Yaskawa INFORM job: tourneTRJ2.JBI

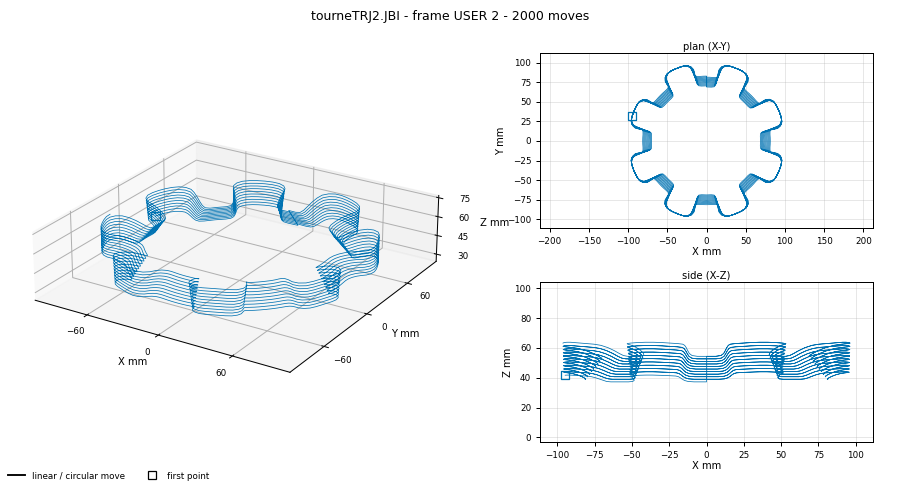
[picture p0: tool path of tourneTRJ2.JBI in frame USER 2, 2000 of 2000 moves have a stored position in this frame; points joined in program order, loops and branches not executed]
/JOB
//NAME tourneTRJ2
///FOLDERNAME DEMO
//POS
///NPOS 2000,0,2000,0,0,0
///USER 2
///TOOL 7
///POSTYPE USER
///RECTAN
///RCONF 1,0,0,0,0,0,0,0,0,0,0,0,0,0,0,0,0,0,0,0,0,0,0,0
C00000=-94.679,31.992,41.678,179.9348,0.0039,-7128.6701
C00001=-93.214,36.189,41.785,179.9926,-0.0033,-7131.2180
C00002=-91.502,40.323,41.785,179.9924,-0.0029,-7133.7821
C00003=-89.570,44.326,41.678,179.9359,-0.0003,-7136.3297
C00004=-87.153,47.905,41.515,178.5880,-0.3682,-7138.7961
C00005=-83.964,50.341,41.355,178.0736,-1.1845,-7140.9450
C00006=-80.606,51.270,41.159,177.8332,-3.2869,-7142.4587
C00007=-77.545,50.645,40.789,178.9173,-3.7322,-7143.1487
C00008=-74.511,49.565,40.048,179.7943,-0.8472,-7143.6320
C00009=-71.724,48.673,39.090,-178.2386,5.1754,-7144.1614
C00010=-69.261,48.447,38.165,-169.6493,15.1644,-7144.9722
C00011=-66.868,49.465,37.495,-147.2874,13.5004,-7146.4919
C00012=-64.059,52.288,37.229,-142.4203,2.3568,-7149.2230
C00013=-61.349,55.398,37.217,-142.1949,-0.1576,-7152.0820
C00014=-58.451,58.451,37.225,-142.2074,0.0000,-7155.0000
C00015=-55.398,61.349,37.217,-142.1949,0.1576,-7157.9180
C00016=-52.288,64.059,37.229,-142.4203,-2.3568,-7160.7770
C00017=-49.465,66.868,37.495,-147.2834,-13.4965,-7163.5081
C00018=-48.447,69.261,38.165,-169.6493,-15.1644,-7165.0278
C00019=-48.673,71.724,39.090,-178.2386,-5.1754,-7165.8386
C00020=-49.565,74.511,40.048,179.7943,0.8472,-7166.3680
C00021=-50.645,77.545,40.789,178.9173,3.7322,-7166.8513
C00022=-51.270,80.606,41.159,177.8332,3.2869,-7167.5413
C00023=-50.341,83.964,41.355,178.0736,1.1845,-7169.0550
C00024=-47.905,87.153,41.515,178.5880,0.3682,-7171.2039
C00025=-44.326,89.570,41.678,179.9359,0.0003,-7173.6703
C00026=-40.323,91.502,41.785,179.9924,0.0029,-7176.2179
C00027=-36.189,93.214,41.785,179.9926,0.0033,-7178.7820
C00028=-31.992,94.679,41.678,179.9348,-0.0039,-7181.3299
C00029=-27.752,95.500,41.515,178.5912,-0.3677,-7183.7963
C00030=-23.775,94.968,41.355,178.0749,-1.1854,-7185.9450
C00031=-20.743,93.250,41.159,177.8320,-3.2854,-7187.4590
C00032=-19.021,90.644,40.789,178.9181,-3.7308,-7188.1488
C00033=-17.640,87.735,40.048,179.7952,-0.8419,-7188.6317
C00034=-16.299,85.134,39.090,-178.2398,5.1751,-7189.1618
C00035=-14.718,83.232,38.165,-169.6494,15.1618,-7189.9720
C00036=-12.305,82.260,37.495,-147.2854,13.4971,-7191.4924
C00037=-8.324,82.270,37.229,-142.4221,2.3584,-7194.2225
C00038=-4.208,82.553,37.217,-142.1936,-0.1593,-7197.0820
C00039=0.000,82.662,37.225,-142.2064,0.0000,-7200.0000
C00040=0.000,81.307,38.958,-141.7572,0.0000,-7200.0000
C00041=4.084,81.202,38.949,-141.7490,0.1755,-7202.8792
C00042=8.115,80.931,38.962,-141.9996,-2.6222,-7205.7259
C00043=12.050,80.963,39.253,-147.5601,-14.5903,-7208.4654
C00044=14.402,82.041,39.987,-171.3983,-14.2979,-7209.9566
C00045=15.932,84.113,41.004,-178.8180,-4.0002,-7210.7254
C00046=17.234,86.943,42.060,179.6316,1.7672,-7211.2119
C00047=18.580,90.119,42.880,178.8638,4.5859,-7211.6495
C00048=20.259,92.987,43.289,177.5830,4.0974,-7212.2909
C00049=23.317,94.913,43.506,177.7331,1.4901,-7213.8024
C00050=27.389,95.566,43.684,178.4237,0.4280,-7215.9922
C00051=31.762,94.755,43.864,179.9221,0.0019,-7218.5312
C00052=36.110,93.244,43.984,179.9872,-0.0012,-7221.1696
C00053=40.400,91.468,43.984,179.9872,-0.0006,-7223.8303
C00054=44.543,89.461,43.864,179.9231,-0.0001,-7226.4689
C00055=48.209,86.942,43.684,178.4246,-0.4305,-7229.0082
C00056=50.626,83.601,43.506,177.7365,-1.4915,-7231.1977
C00057=51.426,80.077,43.289,177.5870,-4.0930,-7232.7089
C00058=50.586,76.861,42.880,178.8633,-4.5829,-7233.3509
C00059=49.291,73.664,42.060,179.6313,-1.7668,-7233.7878
C00060=48.211,70.742,41.004,-178.8201,3.9998,-7234.2746
C00061=47.828,68.195,39.987,-171.4011,14.2972,-7235.0436
C00062=48.729,65.770,39.253,-147.5575,14.5879,-7236.5348
C00063=51.488,62.965,38.962,-141.9986,2.6207,-7239.2737
C00064=54.531,60.307,38.949,-141.7481,-0.1713,-7242.1206
C00065=57.493,57.493,38.958,-141.7571,0.0000,-7245.0000
C00066=60.306,54.531,38.949,-141.7481,0.1717,-7247.8789
C00067=62.965,51.488,38.962,-141.9986,-2.6207,-7250.7263
C00068=65.770,48.729,39.253,-147.5575,-14.5879,-7253.4652
C00069=68.195,47.828,39.987,-171.4011,-14.2972,-7254.9564
C00070=70.742,48.211,41.004,-178.8201,-3.9998,-7255.7254
C00071=73.664,49.291,42.060,179.6313,1.7668,-7256.2122
C00072=76.861,50.586,42.880,178.8633,4.5829,-7256.6491
C00073=80.077,51.426,43.289,177.5870,4.0930,-7257.2911
C00074=83.601,50.626,43.506,177.7365,1.4915,-7258.8023
C00075=86.942,48.209,43.684,178.4246,0.4305,-7260.9918
C00076=89.461,44.543,43.864,179.9231,0.0001,-7263.5311
C00077=91.468,40.400,43.984,179.9872,0.0006,-7266.1697
C00078=93.244,36.110,43.984,179.9872,0.0012,-7268.8304
C00079=94.755,31.762,43.864,179.9221,-0.0019,-7271.4688
C00080=95.566,27.389,43.684,178.4237,-0.4280,-7274.0078
C00081=94.913,23.317,43.506,177.7331,-1.4901,-7276.1976
C00082=92.987,20.259,43.289,177.5830,-4.0974,-7277.7091
C00083=90.119,18.580,42.880,178.8638,-4.5859,-7278.3505
C00084=86.943,17.234,42.060,179.6316,-1.7672,-7278.7881
C00085=84.113,15.932,41.004,-178.8180,4.0002,-7279.2746
C00086=82.041,14.402,39.987,-171.3983,14.2979,-7280.0434
C00087=80.963,12.050,39.253,-147.5601,14.5903,-7281.5346
C00088=80.931,8.115,38.962,-141.9996,2.6222,-7284.2741
C00089=81.202,4.084,38.949,-141.7490,-0.1755,-7287.1208
C00090=81.307,0.000,38.958,-141.7572,-0.0000,-7290.0000
C00091=81.202,-4.084,38.949,-141.7490,0.1755,-7292.8792
C00092=80.931,-8.116,38.962,-141.9996,-2.6227,-7295.7266
C00093=80.963,-12.050,39.253,-147.5601,-14.5903,-7298.4654
C00094=82.041,-14.402,39.987,-171.3983,-14.2979,-7299.9566
C00095=84.113,-15.932,41.004,-178.8180,-4.0002,-7300.7254
C00096=86.943,-17.234,42.060,179.6316,1.7672,-7301.2119
C00097=90.119,-18.580,42.880,178.8638,4.5859,-7301.6495
C00098=92.987,-20.259,43.289,177.5830,4.0974,-7302.2909
C00099=94.913,-23.317,43.506,177.7331,1.4901,-7303.8024
C00100=95.566,-27.389,43.684,178.4237,0.4280,-7305.9922
C00101=94.755,-31.762,43.864,179.9221,0.0019,-7308.5312
C00102=93.244,-36.110,43.984,179.9872,-0.0012,-7311.1696
C00103=91.468,-40.400,43.984,179.9872,-0.0006,-7313.8303
C00104=89.461,-44.543,43.864,179.9231,-0.0001,-7316.4689
C00105=86.942,-48.209,43.684,178.4246,-0.4305,-7319.0082
C00106=83.601,-50.626,43.506,177.7365,-1.4915,-7321.1977
C00107=80.077,-51.426,43.289,177.5870,-4.0930,-7322.7089
C00108=76.861,-50.586,42.880,178.8633,-4.5829,-7323.3509
C00109=73.664,-49.291,42.060,179.6313,-1.7668,-7323.7878
C00110=70.742,-48.211,41.004,-178.8201,3.9998,-7324.2746
C00111=68.195,-47.828,39.987,-171.4011,14.2972,-7325.0436
C00112=65.770,-48.729,39.253,-147.5575,14.5879,-7326.5348
C00113=62.965,-51.488,38.962,-141.9986,2.6207,-7329.2737
C00114=60.307,-54.531,38.949,-141.7481,-0.1713,-7332.1206
C00115=57.493,-57.493,38.958,-141.7571,0.0000,-7335.0000
C00116=54.531,-60.306,38.949,-141.7481,0.1717,-7337.8789
C00117=51.488,-62.965,38.962,-141.9986,-2.6207,-7340.7263
C00118=48.729,-65.770,39.253,-147.5575,-14.5879,-7343.4652
C00119=47.828,-68.195,39.987,-171.4011,-14.2972,-7344.9564
C00120=48.211,-70.742,41.004,-178.8201,-3.9998,-7345.7254
C00121=49.291,-73.664,42.060,179.6313,1.7668,-7346.2122
C00122=50.586,-76.861,42.880,178.8633,4.5829,-7346.6491
C00123=51.426,-80.077,43.289,177.5870,4.0930,-7347.2911
C00124=50.626,-83.601,43.506,177.7365,1.4915,-7348.8023
C00125=48.209,-86.942,43.684,178.4246,0.4305,-7350.9918
C00126=44.543,-89.461,43.864,179.9231,0.0001,-7353.5311
C00127=40.400,-91.468,43.984,179.9872,0.0006,-7356.1697
C00128=36.110,-93.244,43.984,179.9872,0.0012,-7358.8304
C00129=31.762,-94.755,43.864,179.9221,-0.0019,-7361.4688
C00130=27.389,-95.566,43.684,178.4237,-0.4280,-7364.0078
C00131=23.317,-94.913,43.506,177.7331,-1.4901,-7366.1976
C00132=20.259,-92.987,43.289,177.5830,-4.0974,-7367.7091
C00133=18.580,-90.119,42.880,178.8638,-4.5859,-7368.3505
C00134=17.234,-86.943,42.060,179.6316,-1.7672,-7368.7881
C00135=15.932,-84.113,41.004,-178.8180,4.0002,-7369.2746
C00136=14.402,-82.041,39.987,-171.3983,14.2979,-7370.0434
C00137=12.050,-80.963,39.253,-147.5601,14.5903,-7371.5346
C00138=8.115,-80.931,38.962,-141.9996,2.6222,-7374.2741
C00139=4.084,-81.202,38.949,-141.7490,-0.1755,-7377.1208
C00140=0.000,-81.307,38.958,-141.7572,0.0000,-7380.0000
C00141=0.000,-81.307,38.958,-141.7572,0.0000,-7380.0000
C00142=-4.084,-81.202,38.949,-141.7490,0.1755,-7382.8792
C00143=-8.116,-80.931,38.962,-141.9996,-2.6227,-7385.7266
C00144=-12.050,-80.963,39.253,-147.5601,-14.5903,-7388.4654
C00145=-14.402,-82.041,39.987,-171.3983,-14.2979,-7389.9566
C00146=-15.932,-84.113,41.004,-178.8180,-4.0002,-7390.7254
C00147=-17.234,-86.943,42.060,179.6316,1.7672,-7391.2119
C00148=-18.580,-90.119,42.880,178.8638,4.5859,-7391.6495
C00149=-20.259,-92.987,43.289,177.5830,4.0974,-7392.2909
C00150=-23.317,-94.913,43.506,177.7331,1.4901,-7393.8024
C00151=-27.389,-95.566,43.684,178.4237,0.4280,-7395.9922
C00152=-31.762,-94.755,43.864,179.9221,0.0019,-7398.5312
C00153=-36.110,-93.244,43.984,179.9872,-0.0012,-7401.1696
C00154=-40.400,-91.468,43.984,179.9872,-0.0006,-7403.8303
C00155=-44.543,-89.461,43.864,179.9231,-0.0001,-7406.4689
C00156=-48.209,-86.942,43.684,178.4246,-0.4305,-7409.0082
C00157=-50.626,-83.601,43.506,177.7365,-1.4915,-7411.1977
C00158=-51.426,-80.077,43.289,177.5870,-4.0930,-7412.7089
C00159=-50.586,-76.861,42.880,178.8633,-4.5829,-7413.3509
C00160=-49.291,-73.664,42.060,179.6313,-1.7668,-7413.7878
C00161=-48.211,-70.742,41.004,-178.8201,3.9998,-7414.2746
C00162=-47.828,-68.195,39.987,-171.4011,14.2972,-7415.0436
C00163=-48.729,-65.770,39.253,-147.5575,14.5879,-7416.5348
C00164=-51.488,-62.965,38.962,-141.9986,2.6207,-7419.2737
C00165=-54.531,-60.307,38.949,-141.7481,-0.1713,-7422.1206
C00166=-57.493,-57.493,38.958,-141.7571,-0.0000,-7425.0000
C00167=-60.306,-54.531,38.949,-141.7481,0.1717,-7427.8789
C00168=-62.965,-51.488,38.962,-141.9986,-2.6207,-7430.7263
C00169=-65.770,-48.729,39.253,-147.5575,-14.5879,-7433.4652
C00170=-68.195,-47.828,39.987,-171.4011,-14.2972,-7434.9564
C00171=-70.742,-48.211,41.004,-178.8201,-3.9998,-7435.7254
C00172=-73.664,-49.291,42.060,179.6313,1.7668,-7436.2122
C00173=-76.861,-50.586,42.880,178.8633,4.5829,-7436.6491
C00174=-80.077,-51.426,43.289,177.5870,4.0930,-7437.2911
C00175=-83.601,-50.626,43.506,177.7365,1.4915,-7438.8023
C00176=-86.942,-48.209,43.684,178.4246,0.4305,-7440.9918
C00177=-89.461,-44.543,43.864,179.9231,0.0001,-7443.5311
C00178=-91.468,-40.400,43.984,179.9872,0.0006,-7446.1697
C00179=-93.244,-36.110,43.984,179.9872,0.0012,-7448.8304
C00180=-94.755,-31.762,43.864,179.9221,-0.0019,-7451.4688
C00181=-95.566,-27.389,43.684,178.4237,-0.4280,-7454.0078
C00182=-94.913,-23.317,43.506,177.7331,-1.4901,-7456.1976
C00183=-92.987,-20.259,43.289,177.5830,-4.0974,-7457.7091
C00184=-90.119,-18.580,42.880,178.8638,-4.5859,-7458.3505
C00185=-86.943,-17.234,42.060,179.6316,-1.7672,-7458.7881
C00186=-84.113,-15.932,41.004,-178.8180,4.0002,-7459.2746
C00187=-82.041,-14.402,39.987,-171.3983,14.2979,-7460.0434
C00188=-80.963,-12.050,39.253,-147.5601,14.5903,-7461.5346
C00189=-80.931,-8.115,38.962,-141.9996,2.6222,-7464.2741
C00190=-81.202,-4.084,38.949,-141.7490,-0.1755,-7467.1208
C00191=-81.307,0.000,38.958,-141.7572,-0.0000,-7470.0000
C00192=-81.202,4.084,38.949,-141.7490,0.1755,-7472.8792
C00193=-80.931,8.116,38.962,-141.9996,-2.6227,-7475.7266
C00194=-80.963,12.050,39.253,-147.5601,-14.5903,-7478.4654
C00195=-82.041,14.402,39.987,-171.3983,-14.2979,-7479.9566
C00196=-84.113,15.932,41.004,-178.8180,-4.0002,-7480.7254
C00197=-86.943,17.234,42.060,179.6316,1.7672,-7481.2119
C00198=-90.119,18.580,42.880,178.8638,4.5859,-7481.6495
C00199=-92.987,20.259,43.289,177.5830,4.0974,-7482.2909
C00200=-94.913,23.317,43.506,177.7331,1.4901,-7483.8024
C00201=-95.566,27.389,43.684,178.4237,0.4280,-7485.9922
C00202=-94.755,31.762,43.864,179.9221,0.0019,-7488.5312
C00203=-93.244,36.110,43.984,179.9872,-0.0012,-7491.1696
C00204=-91.468,40.400,43.984,179.9872,-0.0006,-7493.8303
C00205=-89.461,44.543,43.864,179.9231,-0.0001,-7496.4689
C00206=-86.942,48.209,43.684,178.4246,-0.4305,-7499.0082
C00207=-83.601,50.626,43.506,177.7365,-1.4915,-7501.1977
C00208=-80.077,51.426,43.289,177.5870,-4.0930,-7502.7089
C00209=-76.861,50.586,42.880,178.8633,-4.5829,-7503.3509
C00210=-73.664,49.291,42.060,179.6313,-1.7668,-7503.7878
C00211=-70.742,48.211,41.004,-178.8201,3.9998,-7504.2746
C00212=-68.195,47.828,39.987,-171.4011,14.2972,-7505.0436
C00213=-65.770,48.729,39.253,-147.5575,14.5879,-7506.5348
C00214=-62.965,51.488,38.962,-141.9986,2.6207,-7509.2737
C00215=-60.307,54.531,38.949,-141.7481,-0.1713,-7512.1206
C00216=-57.493,57.493,38.958,-141.7571,-0.0000,-7515.0000
C00217=-54.531,60.306,38.949,-141.7481,0.1717,-7517.8789
C00218=-51.488,62.965,38.962,-141.9986,-2.6207,-7520.7263
C00219=-48.729,65.770,39.253,-147.5575,-14.5879,-7523.4652
C00220=-47.828,68.195,39.987,-171.4011,-14.2972,-7524.9564
C00221=-48.211,70.742,41.004,-178.8201,-3.9998,-7525.7254
C00222=-49.291,73.664,42.060,179.6313,1.7668,-7526.2122
C00223=-50.586,76.861,42.880,178.8633,4.5829,-7526.6491
C00224=-51.426,80.077,43.289,177.5870,4.0930,-7527.2911
C00225=-50.626,83.601,43.506,177.7365,1.4915,-7528.8023
C00226=-48.209,86.942,43.684,178.4246,0.4305,-7530.9918
C00227=-44.543,89.461,43.864,179.9231,0.0001,-7533.5311
C00228=-40.400,91.468,43.984,179.9872,0.0006,-7536.1697
C00229=-36.110,93.244,43.984,179.9872,0.0012,-7538.8304
C00230=-31.762,94.755,43.864,179.9221,-0.0019,-7541.4688
C00231=-27.389,95.566,43.684,178.4237,-0.4280,-7544.0078
C00232=-23.317,94.913,43.506,177.7331,-1.4901,-7546.1976
C00233=-20.259,92.987,43.289,177.5830,-4.0974,-7547.7091
C00234=-18.580,90.119,42.880,178.8638,-4.5859,-7548.3505
C00235=-17.234,86.943,42.060,179.6316,-1.7672,-7548.7881
C00236=-15.932,84.113,41.004,-178.8180,4.0002,-7549.2746
C00237=-14.402,82.041,39.987,-171.3983,14.2979,-7550.0434
C00238=-12.050,80.963,39.253,-147.5601,14.5903,-7551.5346
C00239=-8.116,80.931,38.962,-141.9996,2.6227,-7554.2734
C00240=-4.084,81.202,38.949,-141.7490,-0.1755,-7557.1208
C00241=0.000,81.307,38.958,-141.7572,-0.0000,-7560.0000
C00242=0.000,79.940,40.681,-141.3939,-0.0000,-7560.0000
C00243=3.959,79.840,40.672,-141.3825,0.1903,-7562.8388
C00244=7.905,79.580,40.686,-141.6632,-2.8895,-7565.6728
C00245=11.791,79.654,41.003,-147.9831,-15.6038,-7568.4202
C00246=14.083,80.839,41.802,-172.9728,-13.2411,-7569.8823
C00247=15.561,83.082,42.912,-179.2626,-2.8848,-7570.6084
C00248=16.825,86.143,44.068,179.5316,2.5969,-7571.0516
C00249=18.134,89.588,44.968,178.8691,5.3340,-7571.4429
C00250=19.771,92.721,45.418,177.4283,4.8395,-7572.0370
C00251=22.856,94.857,45.657,177.4311,1.7993,-7573.5473
C00252=27.022,95.633,45.852,178.2699,0.4949,-7575.7781
C00253=31.529,94.831,46.051,179.9040,0.0017,-7578.3907
C00254=36.031,93.275,46.182,179.9872,-0.0012,-7581.1209
C00255=40.478,91.433,46.182,179.9872,-0.0006,-7583.8793
C00256=44.762,89.350,46.051,179.9026,-0.0025,-7586.6097
C00257=48.515,86.730,45.852,178.2708,-0.4972,-7589.2218
C00258=50.913,83.236,45.657,177.4345,-1.7991,-7591.4529
C00259=51.583,79.544,45.418,177.4322,-4.8395,-7592.9628
C00260=50.526,76.172,44.968,178.8696,-5.3331,-7593.5569
C00261=49.015,72.810,44.068,179.5365,-2.5972,-7593.9481
C00262=47.744,69.752,42.912,-179.2614,2.8847,-7594.3909
C00263=47.203,67.120,41.802,-172.9761,13.2392,-7595.1173
C00264=47.986,64.662,41.003,-147.9821,15.6031,-7596.5793
C00265=50.682,61.862,40.686,-141.6667,2.8929,-7599.3269
C00266=53.655,59.255,40.672,-141.3805,-0.1909,-7602.1606
C00267=56.526,56.526,40.681,-141.3961,0.0000,-7605.0000
C00268=59.255,53.656,40.672,-141.3805,0.1913,-7607.8388
C00269=61.862,50.682,40.686,-141.6667,-2.8929,-7610.6731
C00270=64.662,47.986,41.003,-147.9821,-15.6031,-7613.4207
C00271=67.120,47.203,41.802,-172.9761,-13.2392,-7614.8827
C00272=69.752,47.744,42.912,-179.2614,-2.8847,-7615.6091
C00273=72.810,49.015,44.068,179.5365,2.5972,-7616.0519
C00274=76.172,50.526,44.968,178.8696,5.3331,-7616.4431
C00275=79.544,51.583,45.418,177.4322,4.8395,-7617.0372
C00276=83.236,50.913,45.657,177.4345,1.7991,-7618.5471
C00277=86.730,48.515,45.852,178.2708,0.4972,-7620.7782
C00278=89.350,44.762,46.051,179.9026,0.0025,-7623.3903
C00279=91.433,40.478,46.182,179.9872,0.0006,-7626.1207
C00280=93.275,36.031,46.182,179.9872,0.0012,-7628.8791
C00281=94.831,31.529,46.051,179.9040,-0.0017,-7631.6093
C00282=95.633,27.022,45.852,178.2699,-0.4949,-7634.2219
C00283=94.857,22.856,45.657,177.4311,-1.7993,-7636.4527
C00284=92.721,19.771,45.418,177.4283,-4.8395,-7637.9630
C00285=89.588,18.134,44.968,178.8691,-5.3340,-7638.5571
C00286=86.143,16.825,44.068,179.5316,-2.5969,-7638.9484
C00287=83.082,15.561,42.912,-179.2626,2.8848,-7639.3916
C00288=80.839,14.083,41.802,-172.9728,13.2411,-7640.1177
C00289=79.654,11.791,41.003,-147.9831,15.6038,-7641.5798
C00290=79.580,7.905,40.686,-141.6632,2.8895,-7644.3272
C00291=79.840,3.959,40.672,-141.3825,-0.1903,-7647.1612
C00292=79.940,0.000,40.681,-141.3939,0.0000,-7650.0000
C00293=79.840,-3.959,40.672,-141.3825,0.1903,-7652.8388
C00294=79.580,-7.905,40.686,-141.6677,-2.8888,-7655.6728
C00295=79.654,-11.792,41.003,-147.9832,-15.6042,-7658.4209
C00296=80.839,-14.083,41.802,-172.9728,-13.2411,-7659.8823
C00297=83.082,-15.561,42.912,-179.2626,-2.8848,-7660.6084
C00298=86.143,-16.825,44.068,179.5316,2.5969,-7661.0516
C00299=89.588,-18.134,44.968,178.8691,5.3340,-7661.4429
C00300=92.721,-19.771,45.418,177.4283,4.8395,-7662.0370
C00301=94.857,-22.856,45.657,177.4311,1.7993,-7663.5473
C00302=95.633,-27.022,45.852,178.2699,0.4949,-7665.7781
C00303=94.831,-31.529,46.051,179.9040,0.0017,-7668.3907
C00304=93.275,-36.031,46.182,179.9872,-0.0012,-7671.1209
C00305=91.433,-40.478,46.182,179.9872,-0.0006,-7673.8793
C00306=89.350,-44.762,46.051,179.9026,-0.0025,-7676.6097
C00307=86.730,-48.515,45.852,178.2708,-0.4972,-7679.2218
C00308=83.236,-50.913,45.657,177.4345,-1.7991,-7681.4529
C00309=79.544,-51.583,45.418,177.4322,-4.8395,-7682.9628
C00310=76.172,-50.526,44.968,178.8696,-5.3331,-7683.5569
C00311=72.810,-49.015,44.068,179.5365,-2.5972,-7683.9481
C00312=69.752,-47.744,42.912,-179.2614,2.8847,-7684.3909
C00313=67.120,-47.203,41.802,-172.9761,13.2392,-7685.1173
C00314=64.662,-47.986,41.003,-147.9821,15.6031,-7686.5793
C00315=61.862,-50.682,40.686,-141.6667,2.8929,-7689.3269
C00316=59.255,-53.655,40.672,-141.3805,-0.1909,-7692.1606
C00317=56.526,-56.526,40.681,-141.3961,0.0000,-7695.0000
C00318=53.656,-59.255,40.672,-141.3805,0.1913,-7697.8388
C00319=50.682,-61.862,40.686,-141.6667,-2.8929,-7700.6731
C00320=47.986,-64.662,41.003,-147.9821,-15.6031,-7703.4207
C00321=47.203,-67.120,41.802,-172.9761,-13.2392,-7704.8827
C00322=47.744,-69.752,42.912,-179.2614,-2.8847,-7705.6091
C00323=49.015,-72.810,44.068,179.5365,2.5972,-7706.0519
C00324=50.526,-76.172,44.968,178.8696,5.3331,-7706.4431
C00325=51.583,-79.544,45.418,177.4322,4.8395,-7707.0372
C00326=50.913,-83.236,45.657,177.4345,1.7991,-7708.5471
C00327=48.515,-86.730,45.852,178.2708,0.4972,-7710.7782
C00328=44.762,-89.350,46.051,179.9026,0.0025,-7713.3903
C00329=40.478,-91.433,46.182,179.9872,0.0006,-7716.1207
C00330=36.031,-93.275,46.182,179.9872,0.0012,-7718.8791
C00331=31.529,-94.831,46.051,179.9040,-0.0017,-7721.6093
C00332=27.022,-95.633,45.852,178.2699,-0.4949,-7724.2219
C00333=22.856,-94.857,45.657,177.4311,-1.7993,-7726.4527
C00334=19.771,-92.721,45.418,177.4283,-4.8395,-7727.9630
C00335=18.134,-89.588,44.968,178.8691,-5.3340,-7728.5571
C00336=16.825,-86.143,44.068,179.5316,-2.5969,-7728.9484
C00337=15.561,-83.082,42.912,-179.2626,2.8848,-7729.3916
C00338=14.083,-80.839,41.802,-172.9728,13.2411,-7730.1177
C00339=11.791,-79.654,41.003,-147.9831,15.6038,-7731.5798
C00340=7.905,-79.580,40.686,-141.6632,2.8895,-7734.3272
C00341=3.959,-79.840,40.672,-141.3825,-0.1903,-7737.1612
C00342=0.000,-79.940,40.681,-141.3939,0.0000,-7740.0000
C00343=0.000,-79.940,40.681,-141.3939,0.0000,-7740.0000
C00344=-3.959,-79.840,40.672,-141.3825,0.1903,-7742.8388
C00345=-7.905,-79.580,40.686,-141.6677,-2.8888,-7745.6728
C00346=-11.792,-79.654,41.003,-147.9832,-15.6042,-7748.4209
C00347=-14.083,-80.839,41.802,-172.9728,-13.2411,-7749.8823
C00348=-15.561,-83.082,42.912,-179.2626,-2.8848,-7750.6084
C00349=-16.825,-86.143,44.068,179.5316,2.5969,-7751.0516
C00350=-18.134,-89.588,44.968,178.8691,5.3340,-7751.4429
C00351=-19.771,-92.721,45.418,177.4283,4.8395,-7752.0370
C00352=-22.856,-94.857,45.657,177.4311,1.7993,-7753.5473
C00353=-27.022,-95.633,45.852,178.2699,0.4949,-7755.7781
C00354=-31.529,-94.831,46.051,179.9040,0.0017,-7758.3907
C00355=-36.031,-93.275,46.182,179.9872,-0.0012,-7761.1209
C00356=-40.478,-91.433,46.182,179.9872,-0.0006,-7763.8793
C00357=-44.762,-89.350,46.051,179.9026,-0.0025,-7766.6097
C00358=-48.515,-86.730,45.852,178.2708,-0.4972,-7769.2218
C00359=-50.913,-83.236,45.657,177.4345,-1.7991,-7771.4529
C00360=-51.583,-79.544,45.418,177.4322,-4.8395,-7772.9628
C00361=-50.526,-76.172,44.968,178.8696,-5.3331,-7773.5569
C00362=-49.015,-72.810,44.068,179.5365,-2.5972,-7773.9481
C00363=-47.744,-69.752,42.912,-179.2614,2.8847,-7774.3909
C00364=-47.203,-67.120,41.802,-172.9761,13.2392,-7775.1173
C00365=-47.986,-64.662,41.003,-147.9821,15.6031,-7776.5793
C00366=-50.682,-61.862,40.686,-141.6667,2.8929,-7779.3269
C00367=-53.655,-59.255,40.672,-141.3805,-0.1909,-7782.1606
C00368=-56.526,-56.526,40.681,-141.3961,0.0000,-7785.0000
C00369=-59.255,-53.656,40.672,-141.3805,0.1913,-7787.8388
C00370=-61.862,-50.682,40.686,-141.6667,-2.8929,-7790.6731
C00371=-64.662,-47.986,41.003,-147.9821,-15.6031,-7793.4207
C00372=-67.120,-47.203,41.802,-172.9761,-13.2392,-7794.8827
C00373=-69.752,-47.744,42.912,-179.2614,-2.8847,-7795.6091
C00374=-72.810,-49.015,44.068,179.5365,2.5972,-7796.0519
C00375=-76.172,-50.526,44.968,178.8696,5.3331,-7796.4431
C00376=-79.544,-51.583,45.418,177.4322,4.8395,-7797.0372
C00377=-83.236,-50.913,45.657,177.4345,1.7991,-7798.5471
C00378=-86.730,-48.515,45.852,178.2708,0.4972,-7800.7782
C00379=-89.350,-44.762,46.051,179.9026,0.0025,-7803.3903
C00380=-91.433,-40.478,46.182,179.9872,0.0006,-7806.1207
C00381=-93.275,-36.031,46.182,179.9872,0.0012,-7808.8791
C00382=-94.831,-31.529,46.051,179.9040,-0.0017,-7811.6093
C00383=-95.633,-27.022,45.852,178.2699,-0.4949,-7814.2219
C00384=-94.857,-22.856,45.657,177.4311,-1.7993,-7816.4527
C00385=-92.721,-19.771,45.418,177.4283,-4.8395,-7817.9630
C00386=-89.588,-18.134,44.968,178.8691,-5.3340,-7818.5571
C00387=-86.143,-16.825,44.068,179.5316,-2.5969,-7818.9484
C00388=-83.082,-15.561,42.912,-179.2626,2.8848,-7819.3916
C00389=-80.839,-14.083,41.802,-172.9728,13.2411,-7820.1177
C00390=-79.654,-11.791,41.003,-147.9831,15.6038,-7821.5798
C00391=-79.580,-7.905,40.686,-141.6632,2.8895,-7824.3272
C00392=-79.840,-3.959,40.672,-141.3825,-0.1903,-7827.1612
C00393=-79.940,0.000,40.681,-141.3939,0.0000,-7830.0000
C00394=-79.840,3.959,40.672,-141.3825,0.1903,-7832.8388
C00395=-79.580,7.905,40.686,-141.6677,-2.8888,-7835.6728
C00396=-79.654,11.792,41.003,-147.9832,-15.6042,-7838.4209
C00397=-80.839,14.083,41.802,-172.9728,-13.2411,-7839.8823
C00398=-83.082,15.561,42.912,-179.2626,-2.8848,-7840.6084
C00399=-86.143,16.825,44.068,179.5316,2.5969,-7841.0516
C00400=-89.588,18.134,44.968,178.8691,5.3340,-7841.4429
C00401=-92.721,19.771,45.418,177.4283,4.8395,-7842.0370
C00402=-94.857,22.856,45.657,177.4311,1.7993,-7843.5473
C00403=-95.633,27.022,45.852,178.2699,0.4949,-7845.7781
C00404=-94.831,31.529,46.051,179.9040,0.0017,-7848.3907
C00405=-93.275,36.031,46.182,179.9872,-0.0012,-7851.1209
C00406=-91.433,40.478,46.182,179.9872,-0.0006,-7853.8793
C00407=-89.350,44.762,46.051,179.9026,-0.0025,-7856.6097
C00408=-86.730,48.515,45.852,178.2708,-0.4972,-7859.2218
C00409=-83.236,50.913,45.657,177.4345,-1.7991,-7861.4529
C00410=-79.544,51.583,45.418,177.4322,-4.8395,-7862.9628
C00411=-76.172,50.526,44.968,178.8696,-5.3331,-7863.5569
C00412=-72.810,49.015,44.068,179.5365,-2.5972,-7863.9481
C00413=-69.752,47.744,42.912,-179.2614,2.8847,-7864.3909
C00414=-67.120,47.203,41.802,-172.9761,13.2392,-7865.1173
C00415=-64.662,47.986,41.003,-147.9821,15.6031,-7866.5793
C00416=-61.862,50.682,40.686,-141.6667,2.8929,-7869.3269
C00417=-59.255,53.655,40.672,-141.3805,-0.1909,-7872.1606
C00418=-56.526,56.526,40.681,-141.3961,-0.0000,-7875.0000
C00419=-53.656,59.255,40.672,-141.3805,0.1913,-7877.8388
C00420=-50.682,61.862,40.686,-141.6667,-2.8929,-7880.6731
C00421=-47.986,64.662,41.003,-147.9821,-15.6031,-7883.4207
C00422=-47.203,67.120,41.802,-172.9761,-13.2392,-7884.8827
C00423=-47.744,69.752,42.912,-179.2614,-2.8847,-7885.6091
C00424=-49.015,72.810,44.068,179.5365,2.5972,-7886.0519
C00425=-50.526,76.172,44.968,178.8696,5.3331,-7886.4431
C00426=-51.583,79.544,45.418,177.4322,4.8395,-7887.0372
C00427=-50.913,83.236,45.657,177.4345,1.7991,-7888.5471
C00428=-48.515,86.730,45.852,178.2708,0.4972,-7890.7782
C00429=-44.762,89.350,46.051,179.9026,0.0025,-7893.3903
C00430=-40.478,91.433,46.182,179.9872,0.0006,-7896.1207
C00431=-36.031,93.275,46.182,179.9872,0.0012,-7898.8791
C00432=-31.529,94.831,46.051,179.9040,-0.0017,-7901.6093
C00433=-27.022,95.633,45.852,178.2699,-0.4949,-7904.2219
C00434=-22.856,94.857,45.657,177.4311,-1.7993,-7906.4527
C00435=-19.771,92.721,45.418,177.4283,-4.8395,-7907.9630
C00436=-18.134,89.588,44.968,178.8691,-5.3340,-7908.5571
C00437=-16.825,86.143,44.068,179.5316,-2.5969,-7908.9484
C00438=-15.561,83.082,42.912,-179.2626,2.8848,-7909.3916
C00439=-14.083,80.839,41.802,-172.9728,13.2411,-7910.1177
C00440=-11.792,79.654,41.003,-147.9832,15.6042,-7911.5791
C00441=-7.905,79.580,40.686,-141.6677,2.8888,-7914.3272
C00442=-3.959,79.840,40.672,-141.3825,-0.1903,-7917.1612
C00443=0.000,79.940,40.681,-141.3939,-0.0000,-7920.0000
C00444=0.000,78.562,42.397,-141.1129,-0.0000,-7920.0000
C00445=3.833,78.467,42.387,-141.0976,0.2035,-7922.7966
C00446=7.694,78.220,42.402,-141.4144,-3.1664,-7925.6177
C00447=11.532,78.336,42.745,-148.5477,-16.5332,-7928.3745
C00448=13.762,79.628,43.611,-174.3504,-12.0582,-7929.8055
C00449=15.189,82.045,44.816,-179.5891,-1.8419,-7930.4884
C00450=16.414,85.339,46.074,179.4903,3.3322,-7930.8872
C00451=17.687,89.056,47.055,178.9186,5.9793,-7931.2331
C00452=19.281,92.454,47.546,177.3530,5.5152,-7931.7800
C00453=22.392,94.802,47.807,177.1720,2.1009,-7933.2896
C00454=26.654,95.700,48.020,178.1321,0.5561,-7935.5634
C00455=31.296,94.909,48.237,179.8913,-0.0004,-7938.2498
C00456=35.952,93.306,48.381,179.9872,-0.0012,-7941.0723
C00457=40.555,91.399,48.381,179.9872,-0.0006,-7943.9275
C00458=44.981,89.240,48.237,179.8898,-0.0022,-7946.7502
C00459=48.823,86.517,48.020,178.1320,-0.5583,-7949.4368
C00460=51.201,82.869,47.807,177.1739,-2.0977,-7951.7100
C00461=51.741,79.009,47.546,177.3510,-5.5139,-7953.2198
C00462=50.465,75.478,47.055,178.9198,-5.9790,-7953.7669
C00463=48.737,71.950,46.074,179.4883,-3.3306,-7954.1127
C00464=47.275,68.755,44.816,-179.5904,1.8395,-7954.5119
C00465=46.575,66.037,43.611,-174.3534,12.0585,-7955.1948
C00466=47.238,63.546,42.745,-148.5507,16.5285,-7956.6259
C00467=49.870,60.750,42.402,-141.4112,3.1694,-7959.3828
C00468=52.774,58.195,42.387,-141.0993,-0.2017,-7962.2032
C00469=55.552,55.552,42.397,-141.1143,-0.0000,-7965.0000
C00470=58.195,52.774,42.387,-141.0993,0.2017,-7967.7968
C00471=60.750,49.870,42.402,-141.4147,-3.1690,-7970.6172
C00472=63.546,47.238,42.745,-148.5507,-16.5285,-7973.3741
C00473=66.037,46.575,43.611,-174.3534,-12.0585,-7974.8052
C00474=68.755,47.275,44.816,-179.5904,-1.8395,-7975.4881
C00475=71.950,48.737,46.074,179.4883,3.3306,-7975.8873
C00476=75.478,50.465,47.055,178.9198,5.9790,-7976.2331
C00477=79.009,51.741,47.546,177.3510,5.5139,-7976.7802
C00478=82.869,51.201,47.807,177.1739,2.0977,-7978.2900
C00479=86.517,48.823,48.020,178.1320,0.5583,-7980.5632
C00480=89.240,44.981,48.237,179.8898,0.0022,-7983.2498
C00481=91.399,40.555,48.381,179.9872,0.0006,-7986.0725
C00482=93.306,35.952,48.381,179.9872,0.0012,-7988.9277
C00483=94.909,31.296,48.237,179.8913,0.0004,-7991.7502
C00484=95.700,26.654,48.020,178.1321,-0.5561,-7994.4366
C00485=94.802,22.392,47.807,177.1720,-2.1009,-7996.7104
C00486=92.454,19.281,47.546,177.3530,-5.5152,-7998.2200
C00487=89.056,17.687,47.055,178.9186,-5.9793,-7998.7669
C00488=85.339,16.414,46.074,179.4903,-3.3322,-7999.1128
C00489=82.045,15.189,44.816,-179.5891,1.8419,-7999.5116
C00490=79.628,13.762,43.611,-174.3504,12.0582,-8000.1945
C00491=78.336,11.532,42.745,-148.5477,16.5332,-8001.6255
C00492=78.220,7.694,42.402,-141.4144,3.1664,-8004.3823
C00493=78.467,3.833,42.387,-141.0976,-0.2035,-8007.2034
C00494=78.562,0.000,42.397,-141.1129,-0.0000,-8010.0000
C00495=78.467,-3.833,42.387,-141.0976,0.2035,-8012.7966
C00496=78.220,-7.694,42.402,-141.4184,-3.1733,-8015.6177
C00497=78.336,-11.532,42.745,-148.5477,-16.5332,-8018.3745
C00498=79.628,-13.762,43.611,-174.3504,-12.0582,-8019.8055
C00499=82.045,-15.189,44.816,-179.5891,-1.8419,-8020.4884
C00500=85.339,-16.414,46.074,179.4903,3.3322,-8020.8872
C00501=89.056,-17.687,47.055,178.9186,5.9793,-8021.2331
C00502=92.454,-19.281,47.546,177.3530,5.5152,-8021.7800
C00503=94.802,-22.392,47.807,177.1720,2.1009,-8023.2896
C00504=95.700,-26.654,48.020,178.1321,0.5561,-8025.5634
C00505=94.909,-31.296,48.237,179.8913,-0.0004,-8028.2498
C00506=93.306,-35.952,48.381,179.9872,-0.0012,-8031.0723
C00507=91.399,-40.555,48.381,179.9872,-0.0006,-8033.9275
C00508=89.240,-44.981,48.237,179.8898,-0.0022,-8036.7502
C00509=86.517,-48.823,48.020,178.1320,-0.5583,-8039.4368
C00510=82.869,-51.201,47.807,177.1739,-2.0977,-8041.7100
C00511=79.009,-51.741,47.546,177.3510,-5.5139,-8043.2198
C00512=75.478,-50.465,47.055,178.9198,-5.9790,-8043.7669
C00513=71.950,-48.737,46.074,179.4883,-3.3306,-8044.1127
C00514=68.755,-47.275,44.816,-179.5904,1.8395,-8044.5119
C00515=66.037,-46.575,43.611,-174.3534,12.0585,-8045.1948
C00516=63.546,-47.238,42.745,-148.5507,16.5285,-8046.6259
C00517=60.750,-49.870,42.402,-141.4112,3.1694,-8049.3828
C00518=58.195,-52.774,42.387,-141.0993,-0.2017,-8052.2032
C00519=55.552,-55.552,42.397,-141.1143,-0.0000,-8055.0000
C00520=52.774,-58.195,42.387,-141.0993,0.2017,-8057.7968
C00521=49.870,-60.750,42.402,-141.4147,-3.1690,-8060.6172
C00522=47.238,-63.546,42.745,-148.5507,-16.5285,-8063.3741
C00523=46.575,-66.037,43.611,-174.3534,-12.0585,-8064.8052
C00524=47.275,-68.755,44.816,-179.5904,-1.8395,-8065.4881
C00525=48.737,-71.950,46.074,179.4883,3.3306,-8065.8873
C00526=50.465,-75.478,47.055,178.9198,5.9790,-8066.2331
C00527=51.741,-79.009,47.546,177.3510,5.5139,-8066.7802
C00528=51.201,-82.869,47.807,177.1739,2.0977,-8068.2900
C00529=48.823,-86.517,48.020,178.1320,0.5583,-8070.5632
C00530=44.981,-89.240,48.237,179.8898,0.0022,-8073.2498
C00531=40.555,-91.399,48.381,179.9872,0.0006,-8076.0725
C00532=35.952,-93.306,48.381,179.9872,0.0012,-8078.9277
C00533=31.296,-94.909,48.237,179.8913,0.0004,-8081.7502
C00534=26.654,-95.700,48.020,178.1321,-0.5561,-8084.4366
C00535=22.392,-94.802,47.807,177.1720,-2.1009,-8086.7104
C00536=19.281,-92.454,47.546,177.3530,-5.5152,-8088.2200
C00537=17.687,-89.056,47.055,178.9186,-5.9793,-8088.7669
C00538=16.414,-85.339,46.074,179.4903,-3.3322,-8089.1128
C00539=15.189,-82.045,44.816,-179.5891,1.8419,-8089.5116
C00540=13.762,-79.628,43.611,-174.3504,12.0582,-8090.1945
C00541=11.532,-78.336,42.745,-148.5477,16.5332,-8091.6255
C00542=7.694,-78.220,42.402,-141.4144,3.1664,-8094.3823
C00543=3.833,-78.467,42.387,-141.0976,-0.2035,-8097.2034
C00544=0.000,-78.562,42.397,-141.1129,0.0000,-8100.0000
C00545=0.000,-78.562,42.397,-141.1129,0.0000,-8100.0000
C00546=-3.833,-78.467,42.387,-141.0976,0.2035,-8102.7966
C00547=-7.694,-78.220,42.402,-141.4184,-3.1733,-8105.6177
C00548=-11.532,-78.336,42.745,-148.5477,-16.5332,-8108.3745
C00549=-13.762,-79.628,43.611,-174.3504,-12.0582,-8109.8055
C00550=-15.189,-82.045,44.816,-179.5891,-1.8419,-8110.4884
C00551=-16.414,-85.339,46.074,179.4903,3.3322,-8110.8872
C00552=-17.687,-89.056,47.055,178.9186,5.9793,-8111.2331
C00553=-19.281,-92.454,47.546,177.3530,5.5152,-8111.7800
C00554=-22.392,-94.802,47.807,177.1720,2.1009,-8113.2896
C00555=-26.654,-95.700,48.020,178.1321,0.5561,-8115.5634
C00556=-31.296,-94.909,48.237,179.8913,-0.0004,-8118.2498
C00557=-35.952,-93.306,48.381,179.9872,-0.0012,-8121.0723
C00558=-40.555,-91.399,48.381,179.9872,-0.0006,-8123.9275
C00559=-44.981,-89.240,48.237,179.8898,-0.0022,-8126.7502
C00560=-48.823,-86.517,48.020,178.1320,-0.5583,-8129.4368
C00561=-51.201,-82.869,47.807,177.1739,-2.0977,-8131.7100
C00562=-51.741,-79.009,47.546,177.3510,-5.5139,-8133.2198
C00563=-50.465,-75.478,47.055,178.9198,-5.9790,-8133.7669
C00564=-48.737,-71.950,46.074,179.4883,-3.3306,-8134.1127
C00565=-47.275,-68.755,44.816,-179.5904,1.8395,-8134.5119
C00566=-46.575,-66.037,43.611,-174.3534,12.0585,-8135.1948
C00567=-47.238,-63.546,42.745,-148.5507,16.5285,-8136.6259
C00568=-49.870,-60.750,42.402,-141.4112,3.1694,-8139.3828
C00569=-52.774,-58.195,42.387,-141.0993,-0.2017,-8142.2032
C00570=-55.552,-55.552,42.397,-141.1143,0.0000,-8145.0000
C00571=-58.195,-52.774,42.387,-141.0993,0.2017,-8147.7968
C00572=-60.750,-49.870,42.402,-141.4147,-3.1690,-8150.6172
C00573=-63.546,-47.238,42.745,-148.5507,-16.5285,-8153.3741
C00574=-66.037,-46.575,43.611,-174.3534,-12.0585,-8154.8052
C00575=-68.755,-47.275,44.816,-179.5904,-1.8395,-8155.4881
C00576=-71.950,-48.737,46.074,179.4883,3.3306,-8155.8873
C00577=-75.478,-50.465,47.055,178.9198,5.9790,-8156.2331
C00578=-79.009,-51.741,47.546,177.3510,5.5139,-8156.7802
C00579=-82.869,-51.201,47.807,177.1739,2.0977,-8158.2900
C00580=-86.517,-48.823,48.020,178.1320,0.5583,-8160.5632
C00581=-89.240,-44.981,48.237,179.8898,0.0022,-8163.2498
C00582=-91.399,-40.555,48.381,179.9872,0.0006,-8166.0725
C00583=-93.306,-35.952,48.381,179.9872,0.0012,-8168.9277
C00584=-94.909,-31.296,48.237,179.8913,0.0004,-8171.7502
C00585=-95.700,-26.654,48.020,178.1321,-0.5561,-8174.4366
C00586=-94.802,-22.392,47.807,177.1720,-2.1009,-8176.7104
C00587=-92.454,-19.281,47.546,177.3530,-5.5152,-8178.2200
C00588=-89.056,-17.687,47.055,178.9186,-5.9793,-8178.7669
C00589=-85.339,-16.414,46.074,179.4903,-3.3322,-8179.1128
C00590=-82.045,-15.189,44.816,-179.5891,1.8419,-8179.5116
C00591=-79.628,-13.762,43.611,-174.3504,12.0582,-8180.1945
C00592=-78.336,-11.532,42.745,-148.5477,16.5332,-8181.6255
C00593=-78.220,-7.694,42.402,-141.4144,3.1664,-8184.3823
C00594=-78.467,-3.833,42.387,-141.0976,-0.2035,-8187.2034
C00595=-78.562,0.000,42.397,-141.1129,0.0000,-8190.0000
C00596=-78.467,3.833,42.387,-141.0976,0.2035,-8192.7966
C00597=-78.220,7.694,42.402,-141.4184,-3.1733,-8195.6177
C00598=-78.336,11.532,42.745,-148.5477,-16.5332,-8198.3745
C00599=-79.628,13.762,43.611,-174.3504,-12.0582,-8199.8055
C00600=-82.045,15.189,44.816,-179.5891,-1.8419,-8200.4884
C00601=-85.339,16.414,46.074,179.4903,3.3322,-8200.8872
C00602=-89.056,17.687,47.055,178.9186,5.9793,-8201.2331
C00603=-92.454,19.281,47.546,177.3530,5.5152,-8201.7800
C00604=-94.802,22.392,47.807,177.1720,2.1009,-8203.2896
C00605=-95.700,26.654,48.020,178.1321,0.5561,-8205.5634
C00606=-94.909,31.296,48.237,179.8913,-0.0004,-8208.2498
C00607=-93.306,35.952,48.381,179.9872,-0.0012,-8211.0723
C00608=-91.399,40.555,48.381,179.9872,-0.0006,-8213.9275
C00609=-89.240,44.981,48.237,179.8898,-0.0022,-8216.7502
C00610=-86.517,48.823,48.020,178.1320,-0.5583,-8219.4368
C00611=-82.869,51.201,47.807,177.1739,-2.0977,-8221.7100
C00612=-79.009,51.741,47.546,177.3510,-5.5139,-8223.2198
C00613=-75.478,50.465,47.055,178.9198,-5.9790,-8223.7669
C00614=-71.950,48.737,46.074,179.4883,-3.3306,-8224.1127
C00615=-68.755,47.275,44.816,-179.5904,1.8395,-8224.5119
C00616=-66.037,46.575,43.611,-174.3534,12.0585,-8225.1948
C00617=-63.546,47.238,42.745,-148.5507,16.5285,-8226.6259
C00618=-60.750,49.870,42.402,-141.4112,3.1694,-8229.3828
C00619=-58.195,52.774,42.387,-141.0993,-0.2017,-8232.2032
C00620=-55.552,55.552,42.397,-141.1143,0.0000,-8235.0000
C00621=-52.774,58.195,42.387,-141.0993,0.2017,-8237.7968
C00622=-49.870,60.750,42.402,-141.4147,-3.1690,-8240.6172
C00623=-47.238,63.546,42.745,-148.5507,-16.5285,-8243.3741
C00624=-46.575,66.037,43.611,-174.3534,-12.0585,-8244.8052
C00625=-47.275,68.755,44.816,-179.5904,-1.8395,-8245.4881
C00626=-48.737,71.950,46.074,179.4883,3.3306,-8245.8873
C00627=-50.465,75.478,47.055,178.9198,5.9790,-8246.2331
C00628=-51.741,79.009,47.546,177.3510,5.5139,-8246.7802
C00629=-51.201,82.869,47.807,177.1739,2.0977,-8248.2900
C00630=-48.823,86.517,48.020,178.1320,0.5583,-8250.5632
C00631=-44.981,89.240,48.237,179.8898,0.0022,-8253.2498
C00632=-40.555,91.399,48.381,179.9872,0.0006,-8256.0725
C00633=-35.952,93.306,48.381,179.9872,0.0012,-8258.9277
C00634=-31.296,94.909,48.237,179.8913,0.0004,-8261.7502
C00635=-26.654,95.700,48.020,178.1321,-0.5561,-8264.4366
C00636=-22.392,94.802,47.807,177.1720,-2.1009,-8266.7104
C00637=-19.281,92.454,47.546,177.3530,-5.5152,-8268.2200
C00638=-17.687,89.056,47.055,178.9186,-5.9793,-8268.7669
C00639=-16.414,85.339,46.074,179.4903,-3.3322,-8269.1128
C00640=-15.189,82.045,44.816,-179.5891,1.8419,-8269.5116
C00641=-13.762,79.628,43.611,-174.3504,12.0582,-8270.1945
C00642=-11.532,78.336,42.745,-148.5477,16.5332,-8271.6255
C00643=-7.694,78.220,42.402,-141.4184,3.1733,-8274.3823
C00644=-3.833,78.467,42.387,-141.0976,-0.2035,-8277.2034
C00645=0.000,78.562,42.397,-141.1129,0.0000,-8280.0000
C00646=0.000,77.178,44.107,-140.9053,0.0000,-8280.0000
C00647=3.707,77.088,44.096,-140.8940,0.2219,-8282.7531
C00648=7.481,76.852,44.112,-141.2467,-3.4528,-8285.5598
C00649=11.270,77.011,44.481,-149.2523,-17.3511,-8288.3257
C00650=13.439,78.412,45.416,-175.5313,-10.7991,-8289.7254
C00651=14.814,81.004,46.718,-179.8282,-0.8760,-8290.3637
C00652=16.001,84.532,48.079,179.4791,3.9735,-8290.7187
C00653=17.239,88.522,49.141,178.9964,6.5249,-8291.0200
C00654=18.791,92.187,49.674,177.3355,6.1011,-8291.5211
C00655=21.929,94.746,49.957,176.9535,2.3844,-8293.0317
C00656=26.285,95.767,50.188,178.0119,0.6172,-8295.3479
C00657=31.062,94.986,50.423,179.8804,0.0029,-8298.1086
C00658=35.872,93.336,50.579,179.9872,-0.0012,-8301.0234
C00659=40.633,91.364,50.579,179.9872,-0.0006,-8303.9765
C00660=45.201,89.129,50.423,179.8821,-0.0045,-8306.8914
C00661=49.131,86.304,50.188,178.0134,-0.6169,-8309.6519
C00662=51.489,82.502,49.957,176.9577,-2.3832,-8311.9680
C00663=51.899,78.473,49.674,177.3336,-6.1028,-8313.4791
C00664=50.405,74.784,49.141,178.9911,-6.5252,-8313.9803
C00665=48.459,71.088,48.079,179.4763,-3.9739,-8314.2813
C00666=46.803,67.754,46.718,-179.8313,0.8793,-8314.6359
C00667=45.943,64.949,45.416,-175.5321,10.7985,-8315.2745
C00668=46.486,62.424,44.481,-149.2531,17.3522,-8316.6744
C00669=49.053,59.633,44.112,-141.2455,3.4487,-8319.4401
C00670=51.888,57.130,44.096,-140.8946,-0.2173,-8322.2471
C00671=54.573,54.573,44.107,-140.9054,0.0000,-8325.0000
C00672=57.130,51.888,44.096,-140.8946,0.2173,-8327.7529
C00673=59.633,49.053,44.112,-141.2455,-3.4487,-8330.5599
C00674=62.424,46.486,44.482,-149.2490,-17.3485,-8333.3256
C00675=64.949,45.943,45.416,-175.5321,-10.7985,-8334.7255
C00676=67.754,46.803,46.718,-179.8313,-0.8793,-8335.3641
C00677=71.088,48.459,48.079,179.4763,3.9739,-8335.7187
C00678=74.784,50.405,49.141,178.9911,6.5252,-8336.0197
C00679=78.473,51.899,49.674,177.3336,6.1028,-8336.5209
C00680=82.502,51.489,49.957,176.9577,2.3832,-8338.0320
C00681=86.304,49.131,50.188,178.0134,0.6169,-8340.3481
C00682=89.129,45.201,50.423,179.8821,0.0045,-8343.1086
C00683=91.364,40.633,50.579,179.9872,0.0006,-8346.0235
C00684=93.336,35.872,50.579,179.9872,0.0012,-8348.9766
C00685=94.986,31.062,50.423,179.8804,-0.0029,-8351.8914
C00686=95.767,26.285,50.188,178.0119,-0.6172,-8354.6521
C00687=94.746,21.929,49.957,176.9535,-2.3844,-8356.9683
C00688=92.187,18.791,49.674,177.3355,-6.1011,-8358.4789
C00689=88.522,17.239,49.141,178.9964,-6.5249,-8358.9800
C00690=84.532,16.001,48.079,179.4791,-3.9735,-8359.2813
C00691=81.004,14.814,46.718,-179.8282,0.8760,-8359.6363
C00692=78.412,13.439,45.416,-175.5313,10.7991,-8360.2746
C00693=77.011,11.270,44.481,-149.2523,17.3511,-8361.6743
C00694=76.852,7.481,44.112,-141.2467,3.4528,-8364.4402
C00695=77.088,3.707,44.096,-140.8940,-0.2219,-8367.2469
C00696=77.178,0.000,44.107,-140.9053,-0.0000,-8370.0000
C00697=77.088,-3.707,44.096,-140.8940,0.2219,-8372.7531
C00698=76.852,-7.481,44.112,-141.2467,-3.4528,-8375.5598
C00699=77.011,-11.270,44.482,-149.2523,-17.3511,-8378.3257
C00700=78.412,-13.439,45.416,-175.5313,-10.7991,-8379.7254
C00701=81.004,-14.814,46.718,-179.8282,-0.8760,-8380.3637
C00702=84.532,-16.001,48.079,179.4791,3.9735,-8380.7187
C00703=88.522,-17.239,49.141,178.9964,6.5249,-8381.0200
C00704=92.187,-18.791,49.674,177.3355,6.1011,-8381.5211
C00705=94.746,-21.929,49.957,176.9535,2.3844,-8383.0317
C00706=95.767,-26.285,50.188,178.0119,0.6172,-8385.3479
C00707=94.986,-31.062,50.423,179.8804,0.0029,-8388.1086
C00708=93.336,-35.872,50.579,179.9872,-0.0012,-8391.0234
C00709=91.364,-40.633,50.579,179.9872,-0.0006,-8393.9765
C00710=89.129,-45.201,50.423,179.8821,-0.0045,-8396.8914
C00711=86.304,-49.131,50.188,178.0134,-0.6169,-8399.6519
C00712=82.502,-51.489,49.957,176.9577,-2.3832,-8401.9680
C00713=78.473,-51.899,49.674,177.3336,-6.1028,-8403.4791
C00714=74.784,-50.405,49.141,178.9911,-6.5252,-8403.9803
C00715=71.088,-48.459,48.079,179.4763,-3.9739,-8404.2813
C00716=67.754,-46.803,46.718,-179.8313,0.8793,-8404.6359
C00717=64.949,-45.943,45.416,-175.5321,10.7985,-8405.2745
C00718=62.424,-46.486,44.481,-149.2531,17.3522,-8406.6744
C00719=59.633,-49.053,44.112,-141.2455,3.4487,-8409.4401
C00720=57.130,-51.888,44.096,-140.8946,-0.2173,-8412.2471
C00721=54.573,-54.573,44.107,-140.9054,-0.0000,-8415.0000
C00722=51.888,-57.130,44.096,-140.8946,0.2173,-8417.7529
C00723=49.053,-59.633,44.112,-141.2455,-3.4487,-8420.5599
C00724=46.486,-62.424,44.482,-149.2490,-17.3485,-8423.3256
C00725=45.943,-64.949,45.416,-175.5321,-10.7985,-8424.7255
C00726=46.803,-67.754,46.718,-179.8313,-0.8793,-8425.3641
C00727=48.459,-71.088,48.079,179.4763,3.9739,-8425.7187
C00728=50.405,-74.784,49.141,178.9911,6.5252,-8426.0197
C00729=51.899,-78.473,49.674,177.3336,6.1028,-8426.5209
C00730=51.489,-82.502,49.957,176.9577,2.3832,-8428.0320
C00731=49.131,-86.304,50.188,178.0134,0.6169,-8430.3481
C00732=45.201,-89.129,50.423,179.8821,0.0045,-8433.1086
C00733=40.633,-91.364,50.579,179.9872,0.0006,-8436.0235
C00734=35.872,-93.336,50.579,179.9872,0.0012,-8438.9766
C00735=31.062,-94.986,50.423,179.8804,-0.0029,-8441.8914
C00736=26.285,-95.767,50.188,178.0119,-0.6172,-8444.6521
C00737=21.929,-94.746,49.957,176.9535,-2.3844,-8446.9683
C00738=18.791,-92.187,49.674,177.3355,-6.1011,-8448.4789
C00739=17.239,-88.522,49.141,178.9964,-6.5249,-8448.9800
C00740=16.001,-84.532,48.079,179.4791,-3.9735,-8449.2813
C00741=14.814,-81.004,46.718,-179.8282,0.8760,-8449.6363
C00742=13.439,-78.412,45.416,-175.5313,10.7991,-8450.2746
C00743=11.270,-77.011,44.481,-149.2523,17.3511,-8451.6743
C00744=7.481,-76.852,44.112,-141.2467,3.4528,-8454.4402
C00745=3.707,-77.088,44.096,-140.8940,-0.2219,-8457.2469
C00746=0.000,-77.178,44.107,-140.9053,-0.0000,-8460.0000
C00747=0.000,-77.178,44.107,-140.9053,-0.0000,-8460.0000
C00748=-3.707,-77.088,44.096,-140.8940,0.2219,-8462.7531
C00749=-7.481,-76.852,44.112,-141.2467,-3.4528,-8465.5598
C00750=-11.270,-77.011,44.482,-149.2523,-17.3511,-8468.3257
C00751=-13.439,-78.412,45.416,-175.5313,-10.7991,-8469.7254
C00752=-14.814,-81.004,46.718,-179.8282,-0.8760,-8470.3637
C00753=-16.001,-84.532,48.079,179.4791,3.9735,-8470.7187
C00754=-17.239,-88.522,49.141,178.9964,6.5249,-8471.0200
C00755=-18.791,-92.187,49.674,177.3355,6.1011,-8471.5211
C00756=-21.929,-94.746,49.957,176.9535,2.3844,-8473.0317
C00757=-26.285,-95.767,50.188,178.0119,0.6172,-8475.3479
C00758=-31.062,-94.986,50.423,179.8804,0.0029,-8478.1086
C00759=-35.872,-93.336,50.579,179.9872,-0.0012,-8481.0234
C00760=-40.633,-91.364,50.579,179.9872,-0.0006,-8483.9765
C00761=-45.201,-89.129,50.423,179.8821,-0.0045,-8486.8914
C00762=-49.131,-86.304,50.188,178.0134,-0.6169,-8489.6519
C00763=-51.489,-82.502,49.957,176.9577,-2.3832,-8491.9680
C00764=-51.899,-78.473,49.674,177.3336,-6.1028,-8493.4791
C00765=-50.405,-74.784,49.141,178.9911,-6.5252,-8493.9803
C00766=-48.459,-71.088,48.079,179.4763,-3.9739,-8494.2813
C00767=-46.803,-67.754,46.718,-179.8313,0.8793,-8494.6359
C00768=-45.943,-64.949,45.416,-175.5321,10.7985,-8495.2745
C00769=-46.486,-62.424,44.481,-149.2531,17.3522,-8496.6744
C00770=-49.053,-59.633,44.112,-141.2455,3.4487,-8499.4401
C00771=-51.888,-57.130,44.096,-140.8946,-0.2173,-8502.2471
C00772=-54.573,-54.573,44.107,-140.9054,-0.0000,-8505.0000
C00773=-57.130,-51.888,44.096,-140.8946,0.2173,-8507.7529
C00774=-59.633,-49.053,44.112,-141.2455,-3.4487,-8510.5599
C00775=-62.424,-46.486,44.482,-149.2490,-17.3485,-8513.3256
C00776=-64.949,-45.943,45.416,-175.5321,-10.7985,-8514.7255
C00777=-67.754,-46.803,46.718,-179.8313,-0.8793,-8515.3641
C00778=-71.088,-48.459,48.079,179.4763,3.9739,-8515.7187
C00779=-74.784,-50.405,49.141,178.9911,6.5252,-8516.0197
C00780=-78.473,-51.899,49.674,177.3336,6.1028,-8516.5209
C00781=-82.502,-51.489,49.957,176.9577,2.3832,-8518.0320
C00782=-86.304,-49.131,50.188,178.0134,0.6169,-8520.3481
C00783=-89.129,-45.201,50.423,179.8821,0.0045,-8523.1086
C00784=-91.364,-40.633,50.579,179.9872,0.0006,-8526.0235
C00785=-93.336,-35.872,50.579,179.9872,0.0012,-8528.9766
C00786=-94.986,-31.062,50.423,179.8804,-0.0029,-8531.8914
C00787=-95.767,-26.285,50.188,178.0119,-0.6172,-8534.6521
C00788=-94.746,-21.929,49.957,176.9535,-2.3844,-8536.9683
C00789=-92.187,-18.791,49.674,177.3355,-6.1011,-8538.4789
C00790=-88.522,-17.239,49.141,178.9964,-6.5249,-8538.9800
C00791=-84.532,-16.001,48.079,179.4791,-3.9735,-8539.2813
C00792=-81.004,-14.814,46.718,-179.8282,0.8760,-8539.6363
C00793=-78.412,-13.439,45.416,-175.5313,10.7991,-8540.2746
C00794=-77.011,-11.270,44.481,-149.2523,17.3511,-8541.6743
C00795=-76.852,-7.481,44.112,-141.2467,3.4528,-8544.4402
C00796=-77.088,-3.707,44.096,-140.8940,-0.2219,-8547.2469
C00797=-77.178,0.000,44.107,-140.9053,0.0000,-8550.0000
C00798=-77.088,3.707,44.096,-140.8940,0.2219,-8552.7531
C00799=-76.852,7.481,44.112,-141.2467,-3.4528,-8555.5598
C00800=-77.011,11.270,44.482,-149.2523,-17.3511,-8558.3257
C00801=-78.412,13.439,45.416,-175.5313,-10.7991,-8559.7254
C00802=-81.004,14.814,46.718,-179.8282,-0.8760,-8560.3637
C00803=-84.532,16.001,48.079,179.4791,3.9735,-8560.7187
C00804=-88.522,17.239,49.141,178.9964,6.5249,-8561.0200
C00805=-92.187,18.791,49.674,177.3355,6.1011,-8561.5211
C00806=-94.746,21.929,49.957,176.9535,2.3844,-8563.0317
C00807=-95.767,26.285,50.188,178.0119,0.6172,-8565.3479
C00808=-94.986,31.062,50.423,179.8804,0.0029,-8568.1086
C00809=-93.336,35.872,50.579,179.9872,-0.0012,-8571.0234
C00810=-91.364,40.633,50.579,179.9872,-0.0006,-8573.9765
C00811=-89.129,45.201,50.423,179.8821,-0.0045,-8576.8914
C00812=-86.304,49.131,50.188,178.0134,-0.6169,-8579.6519
C00813=-82.502,51.489,49.957,176.9577,-2.3832,-8581.9680
C00814=-78.473,51.899,49.674,177.3336,-6.1028,-8583.4791
C00815=-74.784,50.405,49.141,178.9911,-6.5252,-8583.9803
C00816=-71.088,48.459,48.079,179.4763,-3.9739,-8584.2813
C00817=-67.754,46.803,46.718,-179.8313,0.8793,-8584.6359
C00818=-64.949,45.943,45.416,-175.5321,10.7985,-8585.2745
C00819=-62.424,46.486,44.481,-149.2531,17.3522,-8586.6744
C00820=-59.633,49.053,44.112,-141.2455,3.4487,-8589.4401
C00821=-57.130,51.888,44.096,-140.8946,-0.2173,-8592.2471
C00822=-54.573,54.573,44.107,-140.9054,0.0000,-8595.0000
C00823=-51.888,57.130,44.096,-140.8946,0.2173,-8597.7529
C00824=-49.053,59.633,44.112,-141.2455,-3.4487,-8600.5599
C00825=-46.486,62.424,44.482,-149.2490,-17.3485,-8603.3256
C00826=-45.943,64.949,45.416,-175.5321,-10.7985,-8604.7255
C00827=-46.803,67.754,46.718,-179.8313,-0.8793,-8605.3641
C00828=-48.459,71.088,48.079,179.4763,3.9739,-8605.7187
C00829=-50.405,74.784,49.141,178.9911,6.5252,-8606.0197
C00830=-51.899,78.473,49.674,177.3336,6.1028,-8606.5209
C00831=-51.489,82.502,49.957,176.9577,2.3832,-8608.0320
C00832=-49.131,86.304,50.188,178.0134,0.6169,-8610.3481
C00833=-45.201,89.129,50.423,179.8821,0.0045,-8613.1086
C00834=-40.633,91.364,50.579,179.9872,0.0006,-8616.0235
C00835=-35.872,93.336,50.579,179.9872,0.0012,-8618.9766
C00836=-31.062,94.986,50.423,179.8804,-0.0029,-8621.8914
C00837=-26.285,95.767,50.188,178.0119,-0.6172,-8624.6521
C00838=-21.929,94.746,49.957,176.9535,-2.3844,-8626.9683
C00839=-18.791,92.187,49.674,177.3355,-6.1011,-8628.4789
C00840=-17.239,88.522,49.141,178.9964,-6.5249,-8628.9800
C00841=-16.001,84.532,48.079,179.4791,-3.9735,-8629.2813
C00842=-14.814,81.004,46.718,-179.8282,0.8760,-8629.6363
C00843=-13.439,78.412,45.416,-175.5313,10.7991,-8630.2746
C00844=-11.270,77.011,44.482,-149.2523,17.3511,-8631.6743
C00845=-7.481,76.852,44.112,-141.2467,3.4528,-8634.4402
C00846=-3.707,77.088,44.096,-140.8940,-0.2219,-8637.2469
C00847=0.000,77.178,44.107,-140.9053,0.0000,-8640.0000
C00848=0.000,75.789,45.812,-140.7711,0.0000,-8640.0000
C00849=3.580,75.703,45.801,-140.7606,0.2311,-8642.7075
C00850=7.267,75.480,45.818,-141.1530,-3.7343,-8645.4993
C00851=11.008,75.681,46.215,-150.0830,-18.0559,-8648.2758
C00852=13.116,77.193,47.218,-176.5222,-9.5058,-8649.6431
C00853=14.439,79.961,48.618,179.9990,-0.0056,-8650.2359
C00854=15.588,83.726,50.084,179.4942,4.5282,-8650.5465
C00855=16.791,87.989,51.229,179.0811,6.9757,-8650.8039
C00856=18.302,91.921,51.802,177.3656,6.6007,-8651.2607
C00857=21.467,94.690,52.107,176.7747,2.6444,-8652.7735
C00858=25.919,95.834,52.356,177.9081,0.6729,-8655.1340
C00859=30.830,95.062,52.610,179.8677,0.0007,-8657.9686
C00860=35.794,93.367,52.777,179.9819,0.0008,-8660.9753
C00861=40.710,91.330,52.777,179.9820,0.0018,-8664.0247
C00862=45.419,89.019,52.610,179.8693,-0.0041,-8667.0314
C00863=49.437,86.092,52.356,177.9051,-0.6676,-8669.8659
C00864=51.776,82.136,52.107,176.7799,-2.6449,-8672.2261
C00865=52.057,77.939,51.802,177.3714,-6.6015,-8673.7397
C00866=50.345,74.091,51.229,179.0848,-6.9720,-8674.1962
C00867=48.181,70.226,50.084,179.4931,-4.5293,-8674.4534
C00868=46.331,66.751,48.618,-179.9967,0.0047,-8674.7640
C00869=45.309,63.858,47.218,-176.5213,9.5073,-8675.3567
C00870=45.731,61.299,46.215,-150.0845,18.0538,-8676.7241
C00871=48.234,58.511,45.818,-141.1526,3.7310,-8679.5007
C00872=50.999,56.061,45.801,-140.7624,-0.2332,-8682.2930
C00873=53.591,53.591,45.812,-140.7695,0.0000,-8685.0000
C00874=56.061,50.999,45.801,-140.7624,0.2332,-8687.7070
C00875=58.511,48.233,45.818,-141.1526,-3.7314,-8690.4999
C00876=61.299,45.731,46.215,-150.0845,-18.0538,-8693.2759
C00877=63.858,45.309,47.218,-176.5213,-9.5073,-8694.6433
C00878=66.751,46.331,48.618,-179.9967,-0.0047,-8695.2360
C00879=70.226,48.181,50.084,179.4931,4.5293,-8695.5466
C00880=74.091,50.345,51.229,179.0848,6.9720,-8695.8038
C00881=77.939,52.057,51.802,177.3714,6.6015,-8696.2603
C00882=82.136,51.776,52.107,176.7799,2.6449,-8697.7739
C00883=86.092,49.437,52.356,177.9051,0.6676,-8700.1341
C00884=89.019,45.419,52.610,179.8693,0.0041,-8702.9686
C00885=91.330,40.710,52.777,179.9820,-0.0018,-8705.9753
C00886=93.367,35.794,52.777,179.9819,-0.0008,-8709.0247
C00887=95.062,30.830,52.610,179.8677,-0.0007,-8712.0314
C00888=95.834,25.919,52.356,177.9081,-0.6729,-8714.8660
C00889=94.690,21.467,52.107,176.7747,-2.6444,-8717.2265
C00890=91.921,18.302,51.802,177.3656,-6.6007,-8718.7393
C00891=87.989,16.791,51.229,179.0811,-6.9757,-8719.1961
C00892=83.726,15.588,50.084,179.4942,-4.5282,-8719.4535
C00893=79.961,14.439,48.618,179.9990,0.0056,-8719.7641
C00894=77.193,13.116,47.218,-176.5222,9.5058,-8720.3569
C00895=75.681,11.008,46.215,-150.0830,18.0559,-8721.7242
C00896=75.480,7.267,45.818,-141.1530,3.7343,-8724.5007
C00897=75.703,3.580,45.801,-140.7606,-0.2311,-8727.2925
C00898=75.789,0.000,45.812,-140.7711,0.0000,-8730.0000
C00899=75.703,-3.580,45.801,-140.7606,0.2311,-8732.7075
C00900=75.480,-7.267,45.818,-141.1530,-3.7343,-8735.4993
C00901=75.681,-11.008,46.215,-150.0830,-18.0559,-8738.2758
C00902=77.193,-13.116,47.218,-176.5222,-9.5058,-8739.6431
C00903=79.961,-14.439,48.618,179.9990,-0.0056,-8740.2359
C00904=83.726,-15.588,50.084,179.4942,4.5282,-8740.5465
C00905=87.989,-16.791,51.229,179.0811,6.9757,-8740.8039
C00906=91.921,-18.302,51.802,177.3656,6.6007,-8741.2607
C00907=94.690,-21.467,52.107,176.7747,2.6444,-8742.7735
C00908=95.834,-25.919,52.356,177.9081,0.6729,-8745.1340
C00909=95.062,-30.830,52.610,179.8677,0.0007,-8747.9686
C00910=93.367,-35.794,52.777,179.9819,0.0008,-8750.9753
C00911=91.330,-40.710,52.777,179.9820,0.0018,-8754.0247
C00912=89.019,-45.419,52.610,179.8693,-0.0041,-8757.0314
C00913=86.092,-49.437,52.356,177.9051,-0.6676,-8759.8659
C00914=82.136,-51.776,52.107,176.7799,-2.6449,-8762.2261
C00915=77.939,-52.057,51.802,177.3714,-6.6015,-8763.7397
C00916=74.091,-50.345,51.229,179.0848,-6.9720,-8764.1962
C00917=70.226,-48.181,50.084,179.4931,-4.5293,-8764.4534
C00918=66.751,-46.331,48.618,-179.9967,0.0047,-8764.7640
C00919=63.858,-45.309,47.218,-176.5213,9.5073,-8765.3567
C00920=61.299,-45.731,46.215,-150.0845,18.0538,-8766.7241
C00921=58.511,-48.234,45.818,-141.1526,3.7310,-8769.5007
C00922=56.061,-50.999,45.801,-140.7624,-0.2332,-8772.2930
C00923=53.591,-53.591,45.812,-140.7695,0.0000,-8775.0000
C00924=50.999,-56.061,45.801,-140.7624,0.2332,-8777.7070
C00925=48.233,-58.511,45.818,-141.1526,-3.7314,-8780.4999
C00926=45.731,-61.299,46.215,-150.0845,-18.0538,-8783.2759
C00927=45.309,-63.858,47.218,-176.5213,-9.5073,-8784.6433
C00928=46.331,-66.751,48.618,-179.9967,-0.0047,-8785.2360
C00929=48.181,-70.226,50.084,179.4931,4.5293,-8785.5466
C00930=50.345,-74.091,51.229,179.0848,6.9720,-8785.8038
C00931=52.057,-77.939,51.802,177.3714,6.6015,-8786.2603
C00932=51.776,-82.136,52.107,176.7799,2.6449,-8787.7739
C00933=49.437,-86.092,52.356,177.9051,0.6676,-8790.1341
C00934=45.419,-89.019,52.610,179.8693,0.0041,-8792.9686
C00935=40.710,-91.330,52.777,179.9820,-0.0018,-8795.9753
C00936=35.794,-93.367,52.777,179.9819,-0.0008,-8799.0247
C00937=30.830,-95.062,52.610,179.8677,-0.0007,-8802.0314
C00938=25.919,-95.834,52.356,177.9081,-0.6729,-8804.8660
C00939=21.467,-94.690,52.107,176.7747,-2.6444,-8807.2265
C00940=18.302,-91.921,51.802,177.3656,-6.6007,-8808.7393
C00941=16.791,-87.989,51.229,179.0811,-6.9757,-8809.1961
C00942=15.588,-83.726,50.084,179.4942,-4.5282,-8809.4535
C00943=14.439,-79.961,48.618,179.9990,0.0056,-8809.7641
C00944=13.116,-77.193,47.218,-176.5222,9.5058,-8810.3569
C00945=11.008,-75.681,46.215,-150.0830,18.0559,-8811.7242
C00946=7.267,-75.480,45.818,-141.1530,3.7343,-8814.5007
C00947=3.580,-75.703,45.801,-140.7606,-0.2311,-8817.2925
C00948=0.000,-75.789,45.812,-140.7711,0.0000,-8820.0000
C00949=0.000,-75.789,45.812,-140.7711,0.0000,-8820.0000
C00950=-3.580,-75.703,45.801,-140.7606,0.2311,-8822.7075
C00951=-7.267,-75.480,45.818,-141.1530,-3.7343,-8825.4993
C00952=-11.008,-75.681,46.215,-150.0830,-18.0559,-8828.2758
C00953=-13.116,-77.193,47.218,-176.5222,-9.5058,-8829.6431
C00954=-14.439,-79.961,48.618,179.9990,-0.0056,-8830.2359
C00955=-15.588,-83.726,50.084,179.4942,4.5282,-8830.5465
C00956=-16.791,-87.989,51.229,179.0811,6.9757,-8830.8039
C00957=-18.302,-91.921,51.802,177.3656,6.6007,-8831.2607
C00958=-21.467,-94.690,52.107,176.7747,2.6444,-8832.7735
C00959=-25.919,-95.834,52.356,177.9081,0.6729,-8835.1340
C00960=-30.830,-95.062,52.610,179.8677,0.0007,-8837.9686
C00961=-35.794,-93.367,52.777,179.9819,0.0008,-8840.9753
C00962=-40.710,-91.330,52.777,179.9820,0.0018,-8844.0247
C00963=-45.419,-89.019,52.610,179.8693,-0.0041,-8847.0314
C00964=-49.437,-86.092,52.356,177.9051,-0.6676,-8849.8659
C00965=-51.776,-82.136,52.107,176.7799,-2.6449,-8852.2261
C00966=-52.057,-77.939,51.802,177.3714,-6.6015,-8853.7397
C00967=-50.345,-74.091,51.229,179.0848,-6.9720,-8854.1962
C00968=-48.181,-70.226,50.084,179.4931,-4.5293,-8854.4534
C00969=-46.331,-66.751,48.618,-179.9967,0.0047,-8854.7640
C00970=-45.309,-63.858,47.218,-176.5213,9.5073,-8855.3567
C00971=-45.731,-61.299,46.215,-150.0845,18.0538,-8856.7241
C00972=-48.234,-58.511,45.818,-141.1526,3.7310,-8859.5007
C00973=-50.999,-56.061,45.801,-140.7624,-0.2332,-8862.2930
C00974=-53.591,-53.591,45.812,-140.7695,-0.0000,-8865.0000
C00975=-56.061,-50.999,45.801,-140.7624,0.2332,-8867.7070
C00976=-58.511,-48.233,45.818,-141.1526,-3.7314,-8870.4999
C00977=-61.299,-45.731,46.215,-150.0845,-18.0538,-8873.2759
C00978=-63.858,-45.309,47.218,-176.5213,-9.5073,-8874.6433
C00979=-66.751,-46.331,48.618,-179.9967,-0.0047,-8875.2360
C00980=-70.226,-48.181,50.084,179.4931,4.5293,-8875.5466
C00981=-74.091,-50.345,51.229,179.0848,6.9720,-8875.8038
C00982=-77.939,-52.057,51.802,177.3714,6.6015,-8876.2603
C00983=-82.136,-51.776,52.107,176.7799,2.6449,-8877.7739
C00984=-86.092,-49.437,52.356,177.9051,0.6676,-8880.1341
C00985=-89.019,-45.419,52.610,179.8693,0.0041,-8882.9686
C00986=-91.330,-40.710,52.777,179.9820,-0.0018,-8885.9753
C00987=-93.367,-35.794,52.777,179.9819,-0.0008,-8889.0247
C00988=-95.062,-30.830,52.610,179.8677,-0.0007,-8892.0314
C00989=-95.834,-25.919,52.356,177.9081,-0.6729,-8894.8660
C00990=-94.690,-21.467,52.107,176.7747,-2.6444,-8897.2265
C00991=-91.921,-18.302,51.802,177.3656,-6.6007,-8898.7393
C00992=-87.989,-16.791,51.229,179.0811,-6.9757,-8899.1961
C00993=-83.726,-15.588,50.084,179.4942,-4.5282,-8899.4535
C00994=-79.961,-14.439,48.618,179.9990,0.0056,-8899.7641
C00995=-77.193,-13.116,47.218,-176.5222,9.5058,-8900.3569
C00996=-75.681,-11.008,46.215,-150.0830,18.0559,-8901.7242
C00997=-75.480,-7.267,45.818,-141.1530,3.7343,-8904.5007
C00998=-75.703,-3.580,45.801,-140.7606,-0.2311,-8907.2925
C00999=-75.789,0.000,45.812,-140.7711,-0.0000,-8910.0000
C01000=-75.703,3.580,45.801,-140.7606,0.2311,-8912.7075
C01001=-75.480,7.267,45.818,-141.1530,-3.7343,-8915.4993
C01002=-75.681,11.008,46.215,-150.0830,-18.0559,-8918.2758
C01003=-77.193,13.116,47.218,-176.5222,-9.5058,-8919.6431
C01004=-79.961,14.439,48.618,179.9990,-0.0056,-8920.2359
C01005=-83.726,15.588,50.084,179.4942,4.5282,-8920.5465
C01006=-87.989,16.791,51.229,179.0811,6.9757,-8920.8039
C01007=-91.921,18.302,51.802,177.3656,6.6007,-8921.2607
C01008=-94.690,21.467,52.107,176.7747,2.6444,-8922.7735
C01009=-95.834,25.919,52.356,177.9081,0.6729,-8925.1340
C01010=-95.062,30.830,52.610,179.8677,0.0007,-8927.9686
C01011=-93.367,35.794,52.777,179.9819,0.0008,-8930.9753
C01012=-91.330,40.710,52.777,179.9820,0.0018,-8934.0247
C01013=-89.019,45.419,52.610,179.8693,-0.0041,-8937.0314
C01014=-86.092,49.437,52.356,177.9051,-0.6676,-8939.8659
C01015=-82.136,51.776,52.107,176.7799,-2.6449,-8942.2261
C01016=-77.939,52.057,51.802,177.3714,-6.6015,-8943.7397
C01017=-74.091,50.345,51.229,179.0848,-6.9720,-8944.1962
C01018=-70.226,48.181,50.084,179.4931,-4.5293,-8944.4534
C01019=-66.751,46.331,48.618,-179.9967,0.0047,-8944.7640
C01020=-63.858,45.309,47.218,-176.5213,9.5073,-8945.3567
C01021=-61.299,45.731,46.215,-150.0845,18.0538,-8946.7241
C01022=-58.511,48.234,45.818,-141.1526,3.7310,-8949.5007
C01023=-56.061,50.999,45.801,-140.7624,-0.2332,-8952.2930
C01024=-53.591,53.591,45.812,-140.7695,-0.0000,-8955.0000
C01025=-50.999,56.061,45.801,-140.7624,0.2332,-8957.7070
C01026=-48.233,58.511,45.818,-141.1526,-3.7314,-8960.4999
C01027=-45.731,61.299,46.215,-150.0845,-18.0538,-8963.2759
C01028=-45.309,63.858,47.218,-176.5213,-9.5073,-8964.6433
C01029=-46.331,66.751,48.618,-179.9967,-0.0047,-8965.2360
C01030=-48.181,70.226,50.084,179.4931,4.5293,-8965.5466
C01031=-50.345,74.091,51.229,179.0848,6.9720,-8965.8038
C01032=-52.057,77.939,51.802,177.3714,6.6015,-8966.2603
C01033=-51.776,82.136,52.107,176.7799,2.6449,-8967.7739
C01034=-49.437,86.092,52.356,177.9051,0.6676,-8970.1341
C01035=-45.419,89.019,52.610,179.8693,0.0041,-8972.9686
C01036=-40.710,91.330,52.777,179.9820,-0.0018,-8975.9753
C01037=-35.794,93.367,52.777,179.9819,-0.0008,-8979.0247
C01038=-30.830,95.062,52.610,179.8677,-0.0007,-8982.0314
C01039=-25.919,95.834,52.356,177.9081,-0.6729,-8984.8660
C01040=-21.467,94.690,52.107,176.7747,-2.6444,-8987.2265
C01041=-18.302,91.921,51.802,177.3656,-6.6007,-8988.7393
C01042=-16.791,87.989,51.229,179.0811,-6.9757,-8989.1961
C01043=-15.588,83.726,50.084,179.4942,-4.5282,-8989.4535
C01044=-14.439,79.961,48.618,179.9990,0.0056,-8989.7641
C01045=-13.116,77.193,47.218,-176.5222,9.5058,-8990.3569
C01046=-11.008,75.681,46.215,-150.0830,18.0559,-8991.7242
C01047=-7.267,75.480,45.818,-141.1530,3.7343,-8994.5007
C01048=-3.580,75.703,45.801,-140.7606,-0.2311,-8997.2925
C01049=0.000,75.789,45.812,-140.7711,-0.0000,-9000.0000
C01050=0.000,74.396,47.516,-140.7138,-0.0000,-9000.0000
C01051=3.453,74.315,47.503,-140.7042,0.2449,-9002.6603
C01052=7.053,74.105,47.522,-141.1410,-4.0170,-9005.4368
C01053=10.745,74.349,47.946,-151.0322,-18.6344,-9008.2235
C01054=12.792,75.972,49.019,-177.3462,-8.2180,-9009.5577
C01055=14.064,78.919,50.519,179.8835,0.7832,-9010.1045
C01056=15.177,82.922,52.090,179.5254,4.9973,-9010.3719
C01057=16.346,87.459,53.317,179.1795,7.3308,-9010.5864
C01058=17.816,91.657,53.931,177.4329,7.0103,-9010.9998
C01059=21.009,94.635,54.258,176.6410,2.8810,-9012.5167
C01060=25.555,95.900,54.525,177.8202,0.7235,-9014.9212
C01061=30.600,95.138,54.796,179.8623,0.0022,-9017.8298
C01062=35.715,93.397,54.976,179.9819,0.0008,-9020.9268
C01063=40.787,91.296,54.976,179.9820,0.0018,-9024.0730
C01064=45.636,88.910,54.796,179.8642,-0.0011,-9027.1707
C01065=49.741,85.881,54.525,177.8219,-0.7191,-9030.0788
C01066=52.061,81.773,54.258,176.6403,-2.8839,-9032.4830
C01067=52.213,77.409,53.931,177.4377,-7.0110,-9034.0000
C01068=50.285,73.401,53.317,179.1794,-7.3322,-9034.4140
C01069=47.903,69.367,52.090,179.5239,-4.9985,-9034.6279
C01070=45.859,65.749,50.519,179.8849,-0.7860,-9034.8952
C01071=44.675,62.766,49.019,-177.3446,8.2234,-9035.4421
C01072=44.975,60.171,47.946,-151.0325,18.6399,-9036.7764
C01073=47.412,57.387,47.522,-141.1396,4.0160,-9039.5628
C01074=50.108,54.990,47.503,-140.7038,-0.2483,-9042.3404
C01075=52.606,52.606,47.516,-140.7163,0.0000,-9045.0000
C01076=54.990,50.108,47.503,-140.7038,0.2483,-9047.6596
C01077=57.387,47.412,47.522,-141.1396,-4.0160,-9050.4372
C01078=60.171,44.975,47.946,-151.0283,-18.6362,-9053.2236
C01079=62.766,44.675,49.019,-177.3446,-8.2234,-9054.5579
C01080=65.749,45.859,50.519,179.8849,0.7860,-9055.1048
C01081=69.367,47.903,52.090,179.5239,4.9985,-9055.3721
C01082=73.401,50.285,53.317,179.1794,7.3322,-9055.5860
C01083=77.409,52.213,53.931,177.4377,7.0110,-9056.0000
C01084=81.773,52.061,54.258,176.6403,2.8839,-9057.5170
C01085=85.881,49.741,54.525,177.8219,0.7191,-9059.9212
C01086=88.910,45.636,54.796,179.8642,0.0011,-9062.8293
C01087=91.296,40.787,54.976,179.9820,-0.0018,-9065.9270
C01088=93.397,35.715,54.976,179.9819,-0.0008,-9069.0732
C01089=95.138,30.600,54.796,179.8623,-0.0022,-9072.1702
C01090=95.900,25.555,54.525,177.8202,-0.7235,-9075.0788
C01091=94.635,21.009,54.258,176.6410,-2.8810,-9077.4833
C01092=91.657,17.816,53.931,177.4329,-7.0103,-9079.0002
C01093=87.459,16.346,53.317,179.1795,-7.3308,-9079.4136
C01094=82.922,15.177,52.090,179.5254,-4.9973,-9079.6281
C01095=78.919,14.064,50.519,179.8835,-0.7832,-9079.8955
C01096=75.972,12.792,49.019,-177.3462,8.2180,-9080.4423
C01097=74.349,10.745,47.946,-151.0322,18.6344,-9081.7765
C01098=74.105,7.053,47.522,-141.1410,4.0170,-9084.5632
C01099=74.315,3.453,47.503,-140.7042,-0.2449,-9087.3397
C01100=74.396,0.000,47.516,-140.7138,0.0000,-9090.0000
C01101=74.315,-3.453,47.503,-140.7042,0.2449,-9092.6603
C01102=74.105,-7.053,47.522,-141.1410,-4.0170,-9095.4368
C01103=74.349,-10.745,47.946,-151.0322,-18.6344,-9098.2235
C01104=75.972,-12.792,49.019,-177.3462,-8.2180,-9099.5577
C01105=78.919,-14.064,50.519,179.8835,0.7832,-9100.1045
C01106=82.922,-15.177,52.090,179.5254,4.9973,-9100.3719
C01107=87.459,-16.346,53.317,179.1795,7.3308,-9100.5864
C01108=91.657,-17.816,53.931,177.4329,7.0103,-9100.9998
C01109=94.635,-21.009,54.258,176.6410,2.8810,-9102.5167
C01110=95.900,-25.555,54.525,177.8202,0.7235,-9104.9212
C01111=95.138,-30.600,54.796,179.8623,0.0022,-9107.8298
C01112=93.397,-35.715,54.976,179.9819,0.0008,-9110.9268
C01113=91.296,-40.787,54.976,179.9820,0.0018,-9114.0730
C01114=88.910,-45.636,54.796,179.8642,-0.0011,-9117.1707
C01115=85.881,-49.741,54.525,177.8219,-0.7191,-9120.0788
C01116=81.773,-52.061,54.258,176.6403,-2.8839,-9122.4830
C01117=77.409,-52.213,53.931,177.4377,-7.0110,-9124.0000
C01118=73.401,-50.285,53.317,179.1794,-7.3322,-9124.4140
C01119=69.367,-47.903,52.090,179.5239,-4.9985,-9124.6279
C01120=65.749,-45.859,50.519,179.8849,-0.7860,-9124.8952
C01121=62.766,-44.675,49.019,-177.3446,8.2234,-9125.4421
C01122=60.171,-44.975,47.946,-151.0325,18.6399,-9126.7764
C01123=57.387,-47.412,47.522,-141.1396,4.0160,-9129.5628
C01124=54.990,-50.108,47.503,-140.7038,-0.2483,-9132.3404
C01125=52.606,-52.606,47.516,-140.7163,0.0000,-9135.0000
C01126=50.108,-54.990,47.503,-140.7038,0.2483,-9137.6596
C01127=47.412,-57.387,47.522,-141.1396,-4.0160,-9140.4372
C01128=44.975,-60.171,47.946,-151.0283,-18.6362,-9143.2236
C01129=44.675,-62.766,49.019,-177.3446,-8.2234,-9144.5579
C01130=45.859,-65.749,50.519,179.8849,0.7860,-9145.1048
C01131=47.903,-69.367,52.090,179.5239,4.9985,-9145.3721
C01132=50.285,-73.401,53.317,179.1794,7.3322,-9145.5860
C01133=52.213,-77.409,53.931,177.4377,7.0110,-9146.0000
C01134=52.061,-81.773,54.258,176.6403,2.8839,-9147.5170
C01135=49.741,-85.881,54.525,177.8219,0.7191,-9149.9212
C01136=45.636,-88.910,54.796,179.8642,0.0011,-9152.8293
C01137=40.787,-91.296,54.976,179.9820,-0.0018,-9155.9270
C01138=35.715,-93.397,54.976,179.9819,-0.0008,-9159.0732
C01139=30.600,-95.138,54.796,179.8623,-0.0022,-9162.1702
C01140=25.555,-95.900,54.525,177.8202,-0.7235,-9165.0788
C01141=21.009,-94.635,54.258,176.6410,-2.8810,-9167.4833
C01142=17.816,-91.657,53.931,177.4329,-7.0103,-9169.0002
C01143=16.346,-87.459,53.317,179.1795,-7.3308,-9169.4136
C01144=15.177,-82.922,52.090,179.5254,-4.9973,-9169.6281
C01145=14.064,-78.919,50.519,179.8835,-0.7832,-9169.8955
C01146=12.792,-75.972,49.019,-177.3462,8.2180,-9170.4423
C01147=10.745,-74.349,47.946,-151.0322,18.6344,-9171.7765
C01148=7.053,-74.105,47.522,-141.1410,4.0170,-9174.5632
C01149=3.453,-74.315,47.503,-140.7042,-0.2449,-9177.3397
C01150=0.000,-74.396,47.516,-140.7138,0.0000,-9180.0000
C01151=0.000,-74.396,47.516,-140.7138,0.0000,-9180.0000
C01152=-3.453,-74.315,47.503,-140.7042,0.2449,-9182.6603
C01153=-7.053,-74.105,47.522,-141.1410,-4.0170,-9185.4368
C01154=-10.745,-74.349,47.946,-151.0322,-18.6344,-9188.2235
C01155=-12.792,-75.972,49.019,-177.3462,-8.2180,-9189.5577
C01156=-14.064,-78.919,50.519,179.8835,0.7832,-9190.1045
C01157=-15.177,-82.922,52.090,179.5254,4.9973,-9190.3719
C01158=-16.346,-87.459,53.317,179.1795,7.3308,-9190.5864
C01159=-17.816,-91.657,53.931,177.4329,7.0103,-9190.9998
C01160=-21.009,-94.635,54.258,176.6410,2.8810,-9192.5167
C01161=-25.555,-95.900,54.525,177.8202,0.7235,-9194.9212
C01162=-30.600,-95.138,54.796,179.8623,0.0022,-9197.8298
C01163=-35.715,-93.397,54.976,179.9819,0.0008,-9200.9268
C01164=-40.787,-91.296,54.976,179.9820,0.0018,-9204.0730
C01165=-45.636,-88.910,54.796,179.8642,-0.0011,-9207.1707
C01166=-49.741,-85.881,54.525,177.8219,-0.7191,-9210.0788
C01167=-52.061,-81.773,54.258,176.6403,-2.8839,-9212.4830
C01168=-52.213,-77.409,53.931,177.4377,-7.0110,-9214.0000
C01169=-50.285,-73.401,53.317,179.1794,-7.3322,-9214.4140
C01170=-47.903,-69.367,52.090,179.5239,-4.9985,-9214.6279
C01171=-45.859,-65.749,50.519,179.8849,-0.7860,-9214.8952
C01172=-44.675,-62.766,49.019,-177.3446,8.2234,-9215.4421
C01173=-44.975,-60.171,47.946,-151.0325,18.6399,-9216.7764
C01174=-47.412,-57.387,47.522,-141.1396,4.0160,-9219.5628
C01175=-50.108,-54.990,47.503,-140.7038,-0.2483,-9222.3404
C01176=-52.606,-52.606,47.516,-140.7163,0.0000,-9225.0000
C01177=-54.990,-50.108,47.503,-140.7038,0.2483,-9227.6596
C01178=-57.387,-47.412,47.522,-141.1396,-4.0160,-9230.4372
C01179=-60.171,-44.975,47.946,-151.0283,-18.6362,-9233.2236
C01180=-62.766,-44.675,49.019,-177.3446,-8.2234,-9234.5579
C01181=-65.749,-45.859,50.519,179.8849,0.7860,-9235.1048
C01182=-69.367,-47.903,52.090,179.5239,4.9985,-9235.3721
C01183=-73.401,-50.285,53.317,179.1794,7.3322,-9235.5860
C01184=-77.409,-52.213,53.931,177.4377,7.0110,-9236.0000
C01185=-81.773,-52.061,54.258,176.6403,2.8839,-9237.5170
C01186=-85.881,-49.741,54.525,177.8219,0.7191,-9239.9212
C01187=-88.910,-45.636,54.796,179.8642,0.0011,-9242.8293
C01188=-91.296,-40.787,54.976,179.9820,-0.0018,-9245.9270
C01189=-93.397,-35.715,54.976,179.9819,-0.0008,-9249.0732
C01190=-95.138,-30.600,54.796,179.8623,-0.0022,-9252.1702
C01191=-95.900,-25.555,54.525,177.8202,-0.7235,-9255.0788
C01192=-94.635,-21.009,54.258,176.6410,-2.8810,-9257.4833
C01193=-91.657,-17.816,53.931,177.4329,-7.0103,-9259.0002
C01194=-87.459,-16.346,53.317,179.1795,-7.3308,-9259.4136
C01195=-82.922,-15.177,52.090,179.5254,-4.9973,-9259.6281
C01196=-78.919,-14.064,50.519,179.8835,-0.7832,-9259.8955
C01197=-75.972,-12.792,49.019,-177.3462,8.2180,-9260.4423
C01198=-74.349,-10.745,47.946,-151.0322,18.6344,-9261.7765
C01199=-74.105,-7.053,47.522,-141.1410,4.0170,-9264.5632
C01200=-74.315,-3.453,47.503,-140.7042,-0.2449,-9267.3397
C01201=-74.396,0.000,47.516,-140.7138,0.0000,-9270.0000
C01202=-74.315,3.453,47.503,-140.7042,0.2449,-9272.6603
C01203=-74.105,7.053,47.522,-141.1410,-4.0170,-9275.4368
C01204=-74.349,10.745,47.946,-151.0322,-18.6344,-9278.2235
C01205=-75.972,12.792,49.019,-177.3462,-8.2180,-9279.5577
C01206=-78.919,14.064,50.519,179.8835,0.7832,-9280.1045
C01207=-82.922,15.177,52.090,179.5254,4.9973,-9280.3719
C01208=-87.459,16.346,53.317,179.1795,7.3308,-9280.5864
C01209=-91.657,17.816,53.931,177.4329,7.0103,-9280.9998
C01210=-94.635,21.009,54.258,176.6410,2.8810,-9282.5167
C01211=-95.900,25.555,54.525,177.8202,0.7235,-9284.9212
C01212=-95.138,30.600,54.796,179.8623,0.0022,-9287.8298
C01213=-93.397,35.715,54.976,179.9819,0.0008,-9290.9268
C01214=-91.296,40.787,54.976,179.9820,0.0018,-9294.0730
C01215=-88.910,45.636,54.796,179.8642,-0.0011,-9297.1707
C01216=-85.881,49.741,54.525,177.8219,-0.7191,-9300.0788
C01217=-81.773,52.061,54.258,176.6403,-2.8839,-9302.4830
C01218=-77.409,52.213,53.931,177.4377,-7.0110,-9304.0000
C01219=-73.401,50.285,53.317,179.1794,-7.3322,-9304.4140
C01220=-69.367,47.903,52.090,179.5239,-4.9985,-9304.6279
C01221=-65.749,45.859,50.519,179.8849,-0.7860,-9304.8952
C01222=-62.766,44.675,49.019,-177.3446,8.2234,-9305.4421
C01223=-60.171,44.975,47.946,-151.0325,18.6399,-9306.7764
C01224=-57.387,47.412,47.522,-141.1396,4.0160,-9309.5628
C01225=-54.990,50.108,47.503,-140.7038,-0.2483,-9312.3404
C01226=-52.606,52.606,47.516,-140.7163,-0.0000,-9315.0000
C01227=-50.108,54.990,47.503,-140.7038,0.2483,-9317.6596
C01228=-47.412,57.387,47.522,-141.1396,-4.0160,-9320.4372
C01229=-44.975,60.171,47.946,-151.0283,-18.6362,-9323.2236
C01230=-44.675,62.766,49.019,-177.3446,-8.2234,-9324.5579
C01231=-45.859,65.749,50.519,179.8849,0.7860,-9325.1048
C01232=-47.903,69.367,52.090,179.5239,4.9985,-9325.3721
C01233=-50.285,73.401,53.317,179.1794,7.3322,-9325.5860
C01234=-52.213,77.409,53.931,177.4377,7.0110,-9326.0000
C01235=-52.061,81.773,54.258,176.6403,2.8839,-9327.5170
C01236=-49.741,85.881,54.525,177.8219,0.7191,-9329.9212
C01237=-45.636,88.910,54.796,179.8642,0.0011,-9332.8293
C01238=-40.787,91.296,54.976,179.9820,-0.0018,-9335.9270
C01239=-35.715,93.397,54.976,179.9819,-0.0008,-9339.0732
C01240=-30.600,95.138,54.796,179.8623,-0.0022,-9342.1702
C01241=-25.555,95.900,54.525,177.8202,-0.7235,-9345.0788
C01242=-21.009,94.635,54.258,176.6410,-2.8810,-9347.4833
C01243=-17.816,91.657,53.931,177.4329,-7.0103,-9349.0002
C01244=-16.346,87.459,53.317,179.1795,-7.3308,-9349.4136
C01245=-15.177,82.922,52.090,179.5254,-4.9973,-9349.6281
C01246=-14.064,78.919,50.519,179.8835,-0.7832,-9349.8955
C01247=-12.792,75.972,49.019,-177.3462,8.2180,-9350.4423
C01248=-10.745,74.349,47.946,-151.0322,18.6344,-9351.7765
C01249=-7.053,74.105,47.522,-141.1410,4.0170,-9354.5632
C01250=-3.453,74.315,47.503,-140.7042,-0.2449,-9357.3397
C01251=0.000,74.396,47.516,-140.7138,-0.0000,-9360.0000
C01252=0.000,73.003,49.219,-140.7299,-0.0000,-9360.0000
C01253=3.325,72.927,49.205,-140.7210,0.2641,-9362.6105
C01254=6.839,72.729,49.225,-141.2026,-4.3012,-9365.3720
C01255=10.483,73.017,49.677,-152.0848,-19.0868,-9368.1701
C01256=12.469,74.753,50.822,-178.0125,-6.9666,-9369.4699
C01257=13.691,77.880,52.422,179.8124,1.4816,-9369.9705
C01258=14.768,82.123,54.099,179.5619,5.3839,-9370.1944
C01259=15.905,86.934,55.407,179.2778,7.6038,-9370.3679
C01260=17.335,91.395,56.062,177.5274,7.3324,-9370.7398
C01261=20.556,94.581,56.410,176.5455,3.0842,-9372.2618
C01262=25.196,95.965,56.695,177.7526,0.7623,-9374.7112
C01263=30.373,95.213,56.983,179.8568,0.0036,-9377.6927
C01264=35.638,93.426,57.174,179.9819,0.0008,-9380.8797
C01265=40.862,91.262,57.174,179.9820,0.0018,-9384.1202
C01266=45.849,88.802,56.983,179.8565,-0.0033,-9387.3076
C01267=50.042,85.674,56.695,177.7539,-0.7661,-9390.2891
C01268=52.343,81.414,56.410,176.5411,-3.0875,-9392.7379
C01269=52.368,76.884,56.062,177.5290,-7.3286,-9394.2600
C01270=50.225,72.718,55.407,179.2794,-7.6004,-9394.6321
C01271=47.627,68.512,54.099,179.5612,-5.3842,-9394.8056
C01272=45.389,64.750,52.422,179.8126,-1.4851,-9395.0300
C01273=44.041,61.675,50.822,-178.0130,6.9633,-9395.5299
C01274=44.219,59.044,49.677,-152.0877,19.0893,-9396.8301
C01275=46.591,56.263,49.225,-141.2030,4.3025,-9399.6279
C01276=49.216,53.919,49.205,-140.7213,-0.2627,-9402.3891
C01277=51.621,51.621,49.219,-140.7299,-0.0000,-9405.0000
C01278=53.919,49.216,49.205,-140.7213,0.2627,-9407.6109
C01279=56.263,46.591,49.225,-141.2030,-4.3025,-9410.3721
C01280=59.044,44.219,49.677,-152.0877,-19.0893,-9413.1699
C01281=61.675,44.041,50.822,-178.0130,-6.9633,-9414.4701
C01282=64.750,45.389,52.422,179.8126,1.4851,-9414.9700
C01283=68.512,47.627,54.099,179.5612,5.3842,-9415.1944
C01284=72.718,50.225,55.407,179.2794,7.6004,-9415.3679
C01285=76.884,52.368,56.062,177.5290,7.3286,-9415.7400
C01286=81.414,52.343,56.410,176.5411,3.0875,-9417.2621
C01287=85.674,50.042,56.695,177.7539,0.7661,-9419.7109
C01288=88.802,45.849,56.983,179.8565,0.0033,-9422.6924
C01289=91.262,40.862,57.174,179.9820,-0.0018,-9425.8798
C01290=93.426,35.638,57.174,179.9819,-0.0008,-9429.1203
C01291=95.213,30.373,56.983,179.8568,-0.0036,-9432.3073
C01292=95.965,25.196,56.695,177.7526,-0.7623,-9435.2888
C01293=94.581,20.556,56.410,176.5455,-3.0842,-9437.7382
C01294=91.395,17.335,56.062,177.5274,-7.3324,-9439.2602
C01295=86.934,15.905,55.407,179.2778,-7.6038,-9439.6321
C01296=82.123,14.768,54.099,179.5619,-5.3839,-9439.8056
C01297=77.880,13.691,52.422,179.8124,-1.4816,-9440.0295
C01298=74.753,12.469,50.822,-178.0125,6.9666,-9440.5301
C01299=73.017,10.483,49.677,-152.0848,19.0868,-9441.8299
C01300=72.729,6.839,49.225,-141.2026,4.3012,-9444.6280
C01301=72.927,3.325,49.205,-140.7210,-0.2641,-9447.3895
C01302=73.003,0.000,49.219,-140.7299,-0.0000,-9450.0000
C01303=72.927,-3.325,49.205,-140.7210,0.2641,-9452.6105
C01304=72.729,-6.839,49.225,-141.2026,-4.3012,-9455.3720
C01305=73.017,-10.483,49.677,-152.0848,-19.0868,-9458.1701
C01306=74.753,-12.469,50.822,-178.0125,-6.9666,-9459.4699
C01307=77.880,-13.691,52.422,179.8124,1.4816,-9459.9705
C01308=82.123,-14.768,54.099,179.5619,5.3839,-9460.1944
C01309=86.934,-15.905,55.407,179.2778,7.6038,-9460.3679
C01310=91.395,-17.335,56.062,177.5274,7.3324,-9460.7398
C01311=94.581,-20.556,56.410,176.5455,3.0842,-9462.2618
C01312=95.965,-25.196,56.695,177.7526,0.7623,-9464.7112
C01313=95.213,-30.373,56.983,179.8568,0.0036,-9467.6927
C01314=93.426,-35.638,57.174,179.9819,0.0008,-9470.8797
C01315=91.262,-40.862,57.174,179.9820,0.0018,-9474.1202
C01316=88.802,-45.849,56.983,179.8565,-0.0033,-9477.3076
C01317=85.674,-50.042,56.695,177.7539,-0.7661,-9480.2891
C01318=81.414,-52.343,56.410,176.5411,-3.0875,-9482.7379
C01319=76.884,-52.368,56.062,177.5290,-7.3286,-9484.2600
C01320=72.718,-50.225,55.407,179.2794,-7.6004,-9484.6321
C01321=68.512,-47.627,54.099,179.5612,-5.3842,-9484.8056
C01322=64.750,-45.389,52.422,179.8126,-1.4851,-9485.0300
C01323=61.675,-44.041,50.822,-178.0130,6.9633,-9485.5299
C01324=59.044,-44.219,49.677,-152.0877,19.0893,-9486.8301
C01325=56.263,-46.591,49.225,-141.2030,4.3025,-9489.6279
C01326=53.919,-49.216,49.205,-140.7213,-0.2627,-9492.3891
C01327=51.621,-51.621,49.219,-140.7299,0.0000,-9495.0000
C01328=49.216,-53.919,49.205,-140.7213,0.2627,-9497.6109
C01329=46.591,-56.263,49.225,-141.2030,-4.3025,-9500.3721
C01330=44.219,-59.044,49.677,-152.0877,-19.0893,-9503.1699
C01331=44.041,-61.675,50.822,-178.0130,-6.9633,-9504.4701
C01332=45.389,-64.750,52.422,179.8126,1.4851,-9504.9700
C01333=47.627,-68.512,54.099,179.5612,5.3842,-9505.1944
C01334=50.225,-72.718,55.407,179.2794,7.6004,-9505.3679
C01335=52.368,-76.884,56.062,177.5290,7.3286,-9505.7400
C01336=52.343,-81.414,56.410,176.5411,3.0875,-9507.2621
C01337=50.042,-85.674,56.695,177.7539,0.7661,-9509.7109
C01338=45.849,-88.802,56.983,179.8565,0.0033,-9512.6924
C01339=40.862,-91.262,57.174,179.9820,-0.0018,-9515.8798
C01340=35.638,-93.426,57.174,179.9819,-0.0008,-9519.1203
C01341=30.373,-95.213,56.983,179.8568,-0.0036,-9522.3073
C01342=25.196,-95.965,56.695,177.7526,-0.7623,-9525.2888
C01343=20.556,-94.581,56.410,176.5455,-3.0842,-9527.7382
C01344=17.335,-91.395,56.062,177.5274,-7.3324,-9529.2602
C01345=15.905,-86.934,55.407,179.2778,-7.6038,-9529.6321
C01346=14.768,-82.123,54.099,179.5619,-5.3839,-9529.8056
C01347=13.691,-77.880,52.422,179.8124,-1.4816,-9530.0295
C01348=12.469,-74.753,50.822,-178.0125,6.9666,-9530.5301
C01349=10.483,-73.017,49.677,-152.0848,19.0868,-9531.8299
C01350=6.839,-72.729,49.225,-141.2026,4.3012,-9534.6280
C01351=3.325,-72.927,49.205,-140.7210,-0.2641,-9537.3895
C01352=0.000,-73.003,49.219,-140.7299,0.0000,-9540.0000
C01353=0.000,-73.003,49.219,-140.7299,0.0000,-9540.0000
C01354=-3.325,-72.927,49.205,-140.7210,0.2641,-9542.6105
C01355=-6.839,-72.729,49.225,-141.2026,-4.3012,-9545.3720
C01356=-10.483,-73.017,49.677,-152.0848,-19.0868,-9548.1701
C01357=-12.469,-74.753,50.822,-178.0125,-6.9666,-9549.4699
C01358=-13.691,-77.880,52.422,179.8124,1.4816,-9549.9705
C01359=-14.768,-82.123,54.099,179.5619,5.3839,-9550.1944
C01360=-15.905,-86.934,55.407,179.2778,7.6038,-9550.3679
C01361=-17.335,-91.395,56.062,177.5274,7.3324,-9550.7398
C01362=-20.556,-94.581,56.410,176.5455,3.0842,-9552.2618
C01363=-25.196,-95.965,56.695,177.7526,0.7623,-9554.7112
C01364=-30.373,-95.213,56.983,179.8568,0.0036,-9557.6927
C01365=-35.638,-93.426,57.174,179.9819,0.0008,-9560.8797
C01366=-40.862,-91.262,57.174,179.9820,0.0018,-9564.1202
C01367=-45.849,-88.802,56.983,179.8565,-0.0033,-9567.3076
C01368=-50.042,-85.674,56.695,177.7539,-0.7661,-9570.2891
C01369=-52.343,-81.414,56.410,176.5411,-3.0875,-9572.7379
C01370=-52.368,-76.884,56.062,177.5290,-7.3286,-9574.2600
C01371=-50.225,-72.718,55.407,179.2794,-7.6004,-9574.6321
C01372=-47.627,-68.512,54.099,179.5612,-5.3842,-9574.8056
C01373=-45.389,-64.750,52.422,179.8126,-1.4851,-9575.0300
C01374=-44.041,-61.675,50.822,-178.0130,6.9633,-9575.5299
C01375=-44.219,-59.044,49.677,-152.0877,19.0893,-9576.8301
C01376=-46.591,-56.263,49.225,-141.2030,4.3025,-9579.6279
C01377=-49.216,-53.919,49.205,-140.7213,-0.2627,-9582.3891
C01378=-51.621,-51.621,49.219,-140.7299,0.0000,-9585.0000
C01379=-53.919,-49.216,49.205,-140.7213,0.2627,-9587.6109
C01380=-56.263,-46.591,49.225,-141.2030,-4.3025,-9590.3721
C01381=-59.044,-44.219,49.677,-152.0877,-19.0893,-9593.1699
C01382=-61.675,-44.041,50.822,-178.0130,-6.9633,-9594.4701
C01383=-64.750,-45.389,52.422,179.8126,1.4851,-9594.9700
C01384=-68.512,-47.627,54.099,179.5612,5.3842,-9595.1944
C01385=-72.718,-50.225,55.407,179.2794,7.6004,-9595.3679
C01386=-76.884,-52.368,56.062,177.5290,7.3286,-9595.7400
C01387=-81.414,-52.343,56.410,176.5411,3.0875,-9597.2621
C01388=-85.674,-50.042,56.695,177.7539,0.7661,-9599.7109
C01389=-88.802,-45.849,56.983,179.8565,0.0033,-9602.6924
C01390=-91.262,-40.862,57.174,179.9820,-0.0018,-9605.8798
C01391=-93.426,-35.638,57.174,179.9819,-0.0008,-9609.1203
C01392=-95.213,-30.373,56.983,179.8568,-0.0036,-9612.3073
C01393=-95.965,-25.196,56.695,177.7526,-0.7623,-9615.2888
C01394=-94.581,-20.556,56.410,176.5455,-3.0842,-9617.7382
C01395=-91.395,-17.335,56.062,177.5274,-7.3324,-9619.2602
C01396=-86.934,-15.905,55.407,179.2778,-7.6038,-9619.6321
C01397=-82.123,-14.768,54.099,179.5619,-5.3839,-9619.8056
C01398=-77.880,-13.691,52.422,179.8124,-1.4816,-9620.0295
C01399=-74.753,-12.469,50.822,-178.0125,6.9666,-9620.5301
C01400=-73.017,-10.483,49.677,-152.0848,19.0868,-9621.8299
C01401=-72.729,-6.839,49.225,-141.2026,4.3012,-9624.6280
C01402=-72.927,-3.325,49.205,-140.7210,-0.2641,-9627.3895
C01403=-73.003,0.000,49.219,-140.7299,0.0000,-9630.0000
C01404=-72.927,3.325,49.205,-140.7210,0.2641,-9632.6105
C01405=-72.729,6.839,49.225,-141.2026,-4.3012,-9635.3720
C01406=-73.017,10.483,49.677,-152.0848,-19.0868,-9638.1701
C01407=-74.753,12.469,50.822,-178.0125,-6.9666,-9639.4699
C01408=-77.880,13.691,52.422,179.8124,1.4816,-9639.9705
C01409=-82.123,14.768,54.099,179.5619,5.3839,-9640.1944
C01410=-86.934,15.905,55.407,179.2778,7.6038,-9640.3679
C01411=-91.395,17.335,56.062,177.5274,7.3324,-9640.7398
C01412=-94.581,20.556,56.410,176.5455,3.0842,-9642.2618
C01413=-95.965,25.196,56.695,177.7526,0.7623,-9644.7112
C01414=-95.213,30.373,56.983,179.8568,0.0036,-9647.6927
C01415=-93.426,35.638,57.174,179.9819,0.0008,-9650.8797
C01416=-91.262,40.862,57.174,179.9820,0.0018,-9654.1202
C01417=-88.802,45.849,56.983,179.8565,-0.0033,-9657.3076
C01418=-85.674,50.042,56.695,177.7539,-0.7661,-9660.2891
C01419=-81.414,52.343,56.410,176.5411,-3.0875,-9662.7379
C01420=-76.884,52.368,56.062,177.5290,-7.3286,-9664.2600
C01421=-72.718,50.225,55.407,179.2794,-7.6004,-9664.6321
C01422=-68.512,47.627,54.099,179.5612,-5.3842,-9664.8056
C01423=-64.750,45.389,52.422,179.8126,-1.4851,-9665.0300
C01424=-61.675,44.041,50.822,-178.0130,6.9633,-9665.5299
C01425=-59.044,44.219,49.677,-152.0877,19.0893,-9666.8301
C01426=-56.263,46.591,49.225,-141.2030,4.3025,-9669.6279
C01427=-53.919,49.216,49.205,-140.7213,-0.2627,-9672.3891
C01428=-51.621,51.621,49.219,-140.7299,0.0000,-9675.0000
C01429=-49.216,53.919,49.205,-140.7213,0.2627,-9677.6109
C01430=-46.591,56.263,49.225,-141.2030,-4.3025,-9680.3721
C01431=-44.219,59.044,49.677,-152.0877,-19.0893,-9683.1699
C01432=-44.041,61.675,50.822,-178.0130,-6.9633,-9684.4701
C01433=-45.389,64.750,52.422,179.8126,1.4851,-9684.9700
C01434=-47.627,68.512,54.099,179.5612,5.3842,-9685.1944
C01435=-50.225,72.718,55.407,179.2794,7.6004,-9685.3679
C01436=-52.368,76.884,56.062,177.5290,7.3286,-9685.7400
C01437=-52.343,81.414,56.410,176.5411,3.0875,-9687.2621
C01438=-50.042,85.674,56.695,177.7539,0.7661,-9689.7109
C01439=-45.849,88.802,56.983,179.8565,0.0033,-9692.6924
C01440=-40.862,91.262,57.174,179.9820,-0.0018,-9695.8798
C01441=-35.638,93.426,57.174,179.9819,-0.0008,-9699.1203
C01442=-30.373,95.213,56.983,179.8568,-0.0036,-9702.3073
C01443=-25.196,95.965,56.695,177.7526,-0.7623,-9705.2888
C01444=-20.556,94.581,56.410,176.5455,-3.0842,-9707.7382
C01445=-17.335,91.395,56.062,177.5274,-7.3324,-9709.2602
C01446=-15.905,86.934,55.407,179.2778,-7.6038,-9709.6321
C01447=-14.768,82.123,54.099,179.5619,-5.3839,-9709.8056
C01448=-13.691,77.880,52.422,179.8124,-1.4816,-9710.0295
C01449=-12.469,74.753,50.822,-178.0125,6.9666,-9710.5301
C01450=-10.483,73.017,49.677,-152.0848,19.0868,-9711.8299
C01451=-6.839,72.729,49.225,-141.2026,4.3012,-9714.6280
C01452=-3.325,72.927,49.205,-140.7210,-0.2641,-9717.3895
C01453=0.000,73.003,49.219,-140.7299,0.0000,-9720.0000
C01454=0.000,71.612,50.923,-140.8239,0.0000,-9720.0000
C01455=3.198,71.541,50.909,-140.8116,0.2724,-9722.5595
C01456=6.625,71.354,50.929,-141.3455,-4.5774,-9725.3045
C01457=10.220,71.688,51.410,-153.2359,-19.4058,-9728.1135
C01458=12.146,73.537,52.627,-178.5505,-5.7667,-9729.3788
C01459=13.319,76.847,54.328,179.7704,2.0988,-9729.8327
C01460=14.363,81.331,56.111,179.6064,5.6993,-9730.0151
C01461=15.469,86.415,57.500,179.3771,7.7949,-9730.1489
C01462=16.861,91.137,58.195,177.6381,7.5640,-9730.4816
C01463=20.110,94.527,58.564,176.4830,3.2557,-9732.0102
C01464=24.842,96.029,58.865,177.7030,0.8018,-9734.5040
C01465=30.149,95.287,59.171,179.8496,-0.0005,-9737.5575
C01466=35.562,93.456,59.373,179.9819,0.0008,-9740.8329
C01467=40.937,91.230,59.373,179.9820,0.0018,-9744.1669
C01468=46.059,88.697,59.171,179.8514,-0.0003,-9747.4422
C01469=50.337,85.469,58.865,177.7073,-0.7986,-9750.4960
C01470=52.621,81.060,58.564,176.4831,-3.2562,-9752.9901
C01471=52.521,76.366,58.195,177.6355,-7.5607,-9754.5184
C01472=50.167,72.043,57.500,179.3759,-7.7906,-9754.8513
C01473=47.354,67.666,56.111,179.6120,-5.6978,-9754.9851
C01474=44.921,63.757,54.328,179.7676,-2.1008,-9755.1672
C01475=43.410,60.587,52.627,-178.5487,5.7649,-9755.6212
C01476=43.464,57.918,51.410,-153.2354,19.4053,-9756.8860
C01477=45.770,55.140,50.929,-141.3424,4.5750,-9759.6950
C01478=48.325,52.849,50.909,-140.8119,-0.2711,-9762.4397
C01479=50.637,50.637,50.923,-140.8226,0.0000,-9765.0000
C01480=52.848,48.326,50.909,-140.8119,0.2720,-9767.5591
C01481=55.140,45.770,50.930,-141.3458,-4.5796,-9770.3050
C01482=57.918,43.464,51.410,-153.2354,-19.4053,-9773.1140
C01483=60.587,43.410,52.627,-178.5487,-5.7649,-9774.3788
C01484=63.757,44.921,54.328,179.7676,2.1008,-9774.8328
C01485=67.666,47.354,56.111,179.6120,5.6978,-9775.0149
C01486=72.043,50.167,57.500,179.3759,7.7906,-9775.1487
C01487=76.366,52.521,58.195,177.6355,7.5607,-9775.4816
C01488=81.060,52.621,58.564,176.4831,3.2562,-9777.0099
C01489=85.469,50.337,58.865,177.7073,0.7986,-9779.5040
C01490=88.697,46.059,59.171,179.8514,0.0003,-9782.5578
C01491=91.230,40.937,59.373,179.9820,-0.0018,-9785.8331
C01492=93.456,35.562,59.373,179.9819,-0.0008,-9789.1671
C01493=95.287,30.149,59.171,179.8496,0.0005,-9792.4425
C01494=96.029,24.842,58.865,177.7030,-0.8018,-9795.4960
C01495=94.527,20.110,58.564,176.4830,-3.2557,-9797.9898
C01496=91.137,16.861,58.195,177.6381,-7.5640,-9799.5184
C01497=86.415,15.469,57.500,179.3771,-7.7949,-9799.8511
C01498=81.331,14.363,56.111,179.6064,-5.6993,-9799.9849
C01499=76.847,13.319,54.328,179.7704,-2.0988,-9800.1673
C01500=73.537,12.146,52.627,-178.5505,5.7667,-9800.6212
C01501=71.688,10.220,51.410,-153.2359,19.4058,-9801.8865
C01502=71.354,6.625,50.929,-141.3455,4.5774,-9804.6955
C01503=71.541,3.198,50.909,-140.8116,-0.2724,-9807.4405
C01504=71.612,0.000,50.923,-140.8239,-0.0000,-9810.0000
C01505=71.541,-3.198,50.909,-140.8116,0.2724,-9812.5595
C01506=71.354,-6.626,50.930,-141.3456,-4.5781,-9815.3053
C01507=71.688,-10.221,51.410,-153.2361,-19.4062,-9818.1143
C01508=73.537,-12.146,52.627,-178.5505,-5.7667,-9819.3788
C01509=76.847,-13.319,54.328,179.7704,2.0988,-9819.8327
C01510=81.331,-14.363,56.111,179.6064,5.6993,-9820.0151
C01511=86.415,-15.469,57.500,179.3771,7.7949,-9820.1489
C01512=91.137,-16.861,58.195,177.6381,7.5640,-9820.4816
C01513=94.527,-20.110,58.564,176.4830,3.2557,-9822.0102
C01514=96.029,-24.842,58.865,177.7030,0.8018,-9824.5040
C01515=95.287,-30.149,59.171,179.8496,-0.0005,-9827.5575
C01516=93.456,-35.562,59.373,179.9819,0.0008,-9830.8329
C01517=91.230,-40.937,59.373,179.9820,0.0018,-9834.1669
C01518=88.697,-46.059,59.171,179.8514,-0.0003,-9837.4422
C01519=85.469,-50.337,58.865,177.7073,-0.7986,-9840.4960
C01520=81.060,-52.621,58.564,176.4831,-3.2562,-9842.9901
C01521=76.366,-52.521,58.195,177.6355,-7.5607,-9844.5184
C01522=72.043,-50.167,57.500,179.3759,-7.7906,-9844.8513
C01523=67.666,-47.354,56.111,179.6120,-5.6978,-9844.9851
C01524=63.757,-44.921,54.328,179.7676,-2.1008,-9845.1672
C01525=60.587,-43.410,52.627,-178.5487,5.7649,-9845.6212
C01526=57.918,-43.464,51.410,-153.2354,19.4053,-9846.8860
C01527=55.140,-45.770,50.929,-141.3424,4.5750,-9849.6950
C01528=52.849,-48.325,50.909,-140.8119,-0.2711,-9852.4397
C01529=50.637,-50.637,50.923,-140.8226,-0.0000,-9855.0000
C01530=48.326,-52.848,50.909,-140.8119,0.2720,-9857.5591
C01531=45.770,-55.140,50.930,-141.3458,-4.5796,-9860.3050
C01532=43.464,-57.918,51.410,-153.2354,-19.4053,-9863.1140
C01533=43.410,-60.587,52.627,-178.5487,-5.7649,-9864.3788
C01534=44.921,-63.757,54.328,179.7676,2.1008,-9864.8328
C01535=47.354,-67.666,56.111,179.6120,5.6978,-9865.0149
C01536=50.167,-72.043,57.500,179.3759,7.7906,-9865.1487
C01537=52.521,-76.366,58.195,177.6355,7.5607,-9865.4816
C01538=52.621,-81.060,58.564,176.4831,3.2562,-9867.0099
C01539=50.337,-85.469,58.865,177.7073,0.7986,-9869.5040
C01540=46.059,-88.697,59.171,179.8514,0.0003,-9872.5578
C01541=40.937,-91.230,59.373,179.9820,-0.0018,-9875.8331
C01542=35.562,-93.456,59.373,179.9819,-0.0008,-9879.1671
C01543=30.149,-95.287,59.171,179.8496,0.0005,-9882.4425
C01544=24.842,-96.029,58.865,177.7030,-0.8018,-9885.4960
C01545=20.110,-94.527,58.564,176.4830,-3.2557,-9887.9898
C01546=16.861,-91.137,58.195,177.6381,-7.5640,-9889.5184
C01547=15.469,-86.415,57.500,179.3771,-7.7949,-9889.8511
C01548=14.363,-81.331,56.111,179.6064,-5.6993,-9889.9849
C01549=13.319,-76.847,54.328,179.7704,-2.0988,-9890.1673
C01550=12.146,-73.537,52.627,-178.5505,5.7667,-9890.6212
C01551=10.220,-71.688,51.410,-153.2359,19.4058,-9891.8865
C01552=6.625,-71.354,50.929,-141.3455,4.5774,-9894.6955
C01553=3.198,-71.541,50.909,-140.8116,-0.2724,-9897.4405
C01554=0.000,-71.612,50.923,-140.8239,-0.0000,-9900.0000
C01555=0.000,-71.612,50.923,-140.8239,-0.0000,-9900.0000
C01556=-3.198,-71.541,50.909,-140.8116,0.2724,-9902.5595
C01557=-6.626,-71.354,50.930,-141.3456,-4.5781,-9905.3053
C01558=-10.221,-71.688,51.410,-153.2361,-19.4062,-9908.1143
C01559=-12.146,-73.537,52.627,-178.5505,-5.7667,-9909.3788
C01560=-13.319,-76.847,54.328,179.7704,2.0988,-9909.8327
C01561=-14.363,-81.331,56.111,179.6064,5.6993,-9910.0151
C01562=-15.469,-86.415,57.500,179.3771,7.7949,-9910.1489
C01563=-16.861,-91.137,58.195,177.6381,7.5640,-9910.4816
C01564=-20.110,-94.527,58.564,176.4830,3.2557,-9912.0102
C01565=-24.842,-96.029,58.865,177.7030,0.8018,-9914.5040
C01566=-30.149,-95.287,59.171,179.8496,-0.0005,-9917.5575
C01567=-35.562,-93.456,59.373,179.9819,0.0008,-9920.8329
C01568=-40.937,-91.230,59.373,179.9820,0.0018,-9924.1669
C01569=-46.059,-88.697,59.171,179.8514,-0.0003,-9927.4422
C01570=-50.337,-85.469,58.865,177.7073,-0.7986,-9930.4960
C01571=-52.621,-81.060,58.564,176.4831,-3.2562,-9932.9901
C01572=-52.521,-76.366,58.195,177.6355,-7.5607,-9934.5184
C01573=-50.167,-72.043,57.500,179.3759,-7.7906,-9934.8513
C01574=-47.354,-67.666,56.111,179.6120,-5.6978,-9934.9851
C01575=-44.921,-63.757,54.328,179.7676,-2.1008,-9935.1672
C01576=-43.410,-60.587,52.627,-178.5487,5.7649,-9935.6212
C01577=-43.464,-57.918,51.410,-153.2354,19.4053,-9936.8860
C01578=-45.770,-55.140,50.929,-141.3424,4.5750,-9939.6950
C01579=-48.325,-52.849,50.909,-140.8119,-0.2711,-9942.4397
C01580=-50.637,-50.637,50.923,-140.8226,-0.0000,-9945.0000
C01581=-52.848,-48.326,50.909,-140.8119,0.2720,-9947.5591
C01582=-55.140,-45.770,50.930,-141.3458,-4.5796,-9950.3050
C01583=-57.918,-43.464,51.410,-153.2354,-19.4053,-9953.1140
C01584=-60.587,-43.410,52.627,-178.5487,-5.7649,-9954.3788
C01585=-63.757,-44.921,54.328,179.7676,2.1008,-9954.8328
C01586=-67.666,-47.354,56.111,179.6120,5.6978,-9955.0149
C01587=-72.043,-50.167,57.500,179.3759,7.7906,-9955.1487
C01588=-76.366,-52.521,58.195,177.6355,7.5607,-9955.4816
C01589=-81.060,-52.621,58.564,176.4831,3.2562,-9957.0099
C01590=-85.469,-50.337,58.865,177.7073,0.7986,-9959.5040
C01591=-88.697,-46.059,59.171,179.8514,0.0003,-9962.5578
C01592=-91.230,-40.937,59.373,179.9820,-0.0018,-9965.8331
C01593=-93.456,-35.562,59.373,179.9819,-0.0008,-9969.1671
C01594=-95.287,-30.149,59.171,179.8496,0.0005,-9972.4425
C01595=-96.029,-24.842,58.865,177.7030,-0.8018,-9975.4960
C01596=-94.527,-20.110,58.564,176.4830,-3.2557,-9977.9898
C01597=-91.137,-16.861,58.195,177.6381,-7.5640,-9979.5184
C01598=-86.415,-15.469,57.500,179.3771,-7.7949,-9979.8511
C01599=-81.331,-14.363,56.111,179.6064,-5.6993,-9979.9849
C01600=-76.847,-13.319,54.328,179.7704,-2.0988,-9980.1673
C01601=-73.537,-12.146,52.627,-178.5505,5.7667,-9980.6212
C01602=-71.688,-10.220,51.410,-153.2359,19.4058,-9981.8865
C01603=-71.354,-6.625,50.929,-141.3455,4.5774,-9984.6955
C01604=-71.541,-3.198,50.909,-140.8116,-0.2724,-9987.4405
C01605=-71.612,0.000,50.923,-140.8239,0.0000,-9990.0000
C01606=-71.541,3.198,50.909,-140.8116,0.2724,-9992.5595
C01607=-71.354,6.626,50.930,-141.3456,-4.5781,-9995.3053
C01608=-71.688,10.221,51.410,-153.2361,-19.4062,-9998.1143
C01609=-73.537,12.146,52.627,-178.5505,-5.7667,-9999.3788
C01610=-76.847,13.319,54.328,179.7704,2.0988,-9999.8327
C01611=-81.331,14.363,56.111,179.6064,5.6993,-10000.0151
C01612=-86.415,15.469,57.500,179.3771,7.7949,-10000.1489
C01613=-91.137,16.861,58.195,177.6381,7.5640,-10000.4816
C01614=-94.527,20.110,58.564,176.4830,3.2557,-10002.0102
C01615=-96.029,24.842,58.865,177.7030,0.8018,-10004.5040
C01616=-95.287,30.149,59.171,179.8496,-0.0005,-10007.5575
C01617=-93.456,35.562,59.373,179.9819,0.0008,-10010.8329
C01618=-91.230,40.937,59.373,179.9820,0.0018,-10014.1669
C01619=-88.697,46.059,59.171,179.8514,-0.0003,-10017.4422
C01620=-85.469,50.337,58.865,177.7073,-0.7986,-10020.4960
C01621=-81.060,52.621,58.564,176.4831,-3.2562,-10022.9901
C01622=-76.366,52.521,58.195,177.6355,-7.5607,-10024.5184
C01623=-72.043,50.167,57.500,179.3759,-7.7906,-10024.8513
C01624=-67.666,47.354,56.111,179.6120,-5.6978,-10024.9851
C01625=-63.757,44.921,54.328,179.7676,-2.1008,-10025.1672
C01626=-60.587,43.410,52.627,-178.5487,5.7649,-10025.6212
C01627=-57.918,43.464,51.410,-153.2354,19.4053,-10026.8860
C01628=-55.140,45.770,50.929,-141.3424,4.5750,-10029.6950
C01629=-52.849,48.325,50.909,-140.8119,-0.2711,-10032.4397
C01630=-50.637,50.637,50.923,-140.8226,0.0000,-10035.0000
C01631=-48.326,52.848,50.909,-140.8119,0.2720,-10037.5591
C01632=-45.770,55.140,50.930,-141.3458,-4.5796,-10040.3050
C01633=-43.464,57.918,51.410,-153.2354,-19.4053,-10043.1140
C01634=-43.410,60.587,52.627,-178.5487,-5.7649,-10044.3788
C01635=-44.921,63.757,54.328,179.7676,2.1008,-10044.8328
C01636=-47.354,67.666,56.111,179.6120,5.6978,-10045.0149
C01637=-50.167,72.043,57.500,179.3759,7.7906,-10045.1487
C01638=-52.521,76.366,58.195,177.6355,7.5607,-10045.4816
C01639=-52.621,81.060,58.564,176.4831,3.2562,-10047.0099
C01640=-50.337,85.469,58.865,177.7073,0.7986,-10049.5040
C01641=-46.059,88.697,59.171,179.8514,0.0003,-10052.5578
C01642=-40.937,91.230,59.373,179.9820,-0.0018,-10055.8331
C01643=-35.562,93.456,59.373,179.9819,-0.0008,-10059.1671
C01644=-30.149,95.287,59.171,179.8496,0.0005,-10062.4425
C01645=-24.842,96.029,58.865,177.7030,-0.8018,-10065.4960
C01646=-20.110,94.527,58.564,176.4830,-3.2557,-10067.9898
C01647=-16.861,91.137,58.195,177.6381,-7.5640,-10069.5184
C01648=-15.469,86.415,57.500,179.3771,-7.7949,-10069.8511
C01649=-14.363,81.331,56.111,179.6064,-5.6993,-10069.9849
C01650=-13.319,76.847,54.328,179.7704,-2.0988,-10070.1673
C01651=-12.146,73.537,52.627,-178.5505,5.7667,-10070.6212
C01652=-10.221,71.688,51.410,-153.2361,19.4062,-10071.8857
C01653=-6.626,71.354,50.930,-141.3456,4.5781,-10074.6947
C01654=-3.198,71.541,50.909,-140.8116,-0.2724,-10077.4405
C01655=0.000,71.612,50.923,-140.8239,0.0000,-10080.0000
C01656=0.000,70.224,52.630,-140.9867,0.0000,-10080.0000
C01657=3.072,70.158,52.615,-140.9755,0.2846,-10082.5072
C01658=6.412,69.984,52.637,-141.5661,-4.8461,-10085.2349
C01659=9.959,70.362,53.146,-154.4717,-19.5944,-10088.0561
C01660=11.825,72.328,54.436,-178.9707,-4.6321,-10089.2852
C01661=12.951,75.822,56.240,179.7522,2.6357,-10089.6930
C01662=13.963,80.549,58.128,179.6532,5.9380,-10089.8344
C01663=15.041,85.905,59.597,179.4669,7.9061,-10089.9312
C01664=16.396,90.884,60.330,177.7605,7.7070,-10090.2265
C01665=19.672,94.474,60.719,176.4586,3.3893,-10091.7624
C01666=24.496,96.092,61.037,177.6795,0.8285,-10094.3014
C01667=29.931,95.359,61.359,179.8441,0.0009,-10097.4259
C01668=35.488,93.484,61.571,179.9819,0.0007,-10100.7876
C01669=41.009,91.197,61.571,179.9820,0.0018,-10104.2123
C01670=46.265,88.593,61.359,179.8436,-0.0024,-10107.5744
C01671=50.626,85.269,61.037,177.6762,-0.8270,-10110.6985
C01672=52.893,80.714,60.719,176.4619,-3.3877,-10113.2374
C01673=52.671,75.858,60.330,177.7582,-7.7084,-10114.7737
C01674=50.109,71.379,59.597,179.4666,-7.9076,-10115.0694
C01675=47.084,66.830,58.128,179.6563,-5.9377,-10115.1660
C01676=44.457,62.772,56.240,179.7505,-2.6330,-10115.3073
C01677=42.782,59.505,54.436,-178.9712,4.6316,-10115.7148
C01678=42.712,56.796,53.146,-154.4681,19.5904,-10116.9441
C01679=44.952,54.020,52.637,-141.5644,4.8467,-10119.7651
C01680=47.437,51.781,52.615,-140.9755,-0.2845,-10122.4931
C01681=49.656,49.656,52.630,-140.9851,-0.0052,-10125.0000
C01682=51.781,47.437,52.615,-140.9755,0.2845,-10127.5069
C01683=54.020,44.952,52.637,-141.5644,-4.8467,-10130.2349
C01684=56.796,42.711,53.146,-154.4683,-19.5906,-10133.0566
C01685=59.505,42.782,54.436,-178.9712,-4.6316,-10134.2852
C01686=62.772,44.457,56.240,179.7505,2.6330,-10134.6927
C01687=66.830,47.084,58.128,179.6563,5.9377,-10134.8340
C01688=71.379,50.109,59.597,179.4666,7.9076,-10134.9306
C01689=75.858,52.671,60.330,177.7582,7.7084,-10135.2263
C01690=80.714,52.893,60.719,176.4619,3.3877,-10136.7626
C01691=85.269,50.626,61.037,177.6762,0.8270,-10139.3015
C01692=88.593,46.265,61.359,179.8436,0.0024,-10142.4256
C01693=91.197,41.009,61.571,179.9820,-0.0018,-10145.7877
C01694=93.484,35.488,61.571,179.9819,-0.0007,-10149.2124
C01695=95.359,29.931,61.359,179.8441,-0.0009,-10152.5741
C01696=96.092,24.496,61.037,177.6795,-0.8285,-10155.6986
C01697=94.474,19.672,60.719,176.4586,-3.3893,-10158.2376
C01698=90.884,16.396,60.330,177.7605,-7.7070,-10159.7735
C01699=85.905,15.041,59.597,179.4669,-7.9061,-10160.0688
C01700=80.549,13.963,58.128,179.6532,-5.9380,-10160.1656
C01701=75.822,12.951,56.240,179.7522,-2.6357,-10160.3070
C01702=72.328,11.825,54.436,-178.9707,4.6321,-10160.7148
C01703=70.362,9.959,53.146,-154.4717,19.5944,-10161.9439
C01704=69.984,6.412,52.637,-141.5661,4.8461,-10164.7651
C01705=70.158,3.072,52.615,-140.9755,-0.2846,-10167.4928
C01706=70.224,0.000,52.630,-140.9867,0.0000,-10170.0000
C01707=70.158,-3.071,52.615,-140.9755,0.2852,-10172.5064
C01708=69.984,-6.412,52.637,-141.5661,-4.8461,-10175.2349
C01709=70.362,-9.959,53.146,-154.4655,-19.5894,-10178.0561
C01710=72.328,-11.825,54.436,-178.9707,-4.6321,-10179.2852
C01711=75.822,-12.951,56.240,179.7522,2.6357,-10179.6930
C01712=80.549,-13.963,58.128,179.6532,5.9380,-10179.8344
C01713=85.905,-15.041,59.597,179.4669,7.9061,-10179.9312
C01714=90.884,-16.396,60.330,177.7605,7.7070,-10180.2265
C01715=94.474,-19.672,60.719,176.4586,3.3893,-10181.7624
C01716=96.092,-24.496,61.037,177.6795,0.8285,-10184.3014
C01717=95.359,-29.931,61.359,179.8441,0.0009,-10187.4259
C01718=93.484,-35.488,61.571,179.9819,0.0007,-10190.7876
C01719=91.197,-41.009,61.571,179.9820,0.0018,-10194.2123
C01720=88.593,-46.265,61.359,179.8436,-0.0024,-10197.5744
C01721=85.269,-50.626,61.037,177.6762,-0.8270,-10200.6985
C01722=80.714,-52.893,60.719,176.4619,-3.3877,-10203.2374
C01723=75.858,-52.671,60.330,177.7582,-7.7084,-10204.7737
C01724=71.379,-50.109,59.597,179.4666,-7.9076,-10205.0694
C01725=66.830,-47.084,58.128,179.6563,-5.9377,-10205.1660
C01726=62.772,-44.457,56.240,179.7505,-2.6330,-10205.3073
C01727=59.505,-42.782,54.436,-178.9712,4.6316,-10205.7148
C01728=56.796,-42.712,53.146,-154.4681,19.5904,-10206.9441
C01729=54.020,-44.952,52.637,-141.5644,4.8467,-10209.7651
C01730=51.781,-47.437,52.615,-140.9755,-0.2845,-10212.4931
C01731=49.656,-49.656,52.630,-140.9851,-0.0052,-10215.0000
C01732=47.437,-51.781,52.615,-140.9755,0.2845,-10217.5069
C01733=44.952,-54.020,52.637,-141.5644,-4.8467,-10220.2349
C01734=42.711,-56.796,53.146,-154.4683,-19.5906,-10223.0566
C01735=42.782,-59.505,54.436,-178.9712,-4.6316,-10224.2852
C01736=44.457,-62.772,56.240,179.7505,2.6330,-10224.6927
C01737=47.084,-66.830,58.128,179.6563,5.9377,-10224.8340
C01738=50.109,-71.379,59.597,179.4666,7.9076,-10224.9306
C01739=52.671,-75.858,60.330,177.7582,7.7084,-10225.2263
C01740=52.893,-80.714,60.719,176.4619,3.3877,-10226.7626
C01741=50.626,-85.269,61.037,177.6762,0.8270,-10229.3015
C01742=46.265,-88.593,61.359,179.8436,0.0024,-10232.4256
C01743=41.009,-91.197,61.571,179.9820,-0.0018,-10235.7877
C01744=35.488,-93.484,61.571,179.9819,-0.0007,-10239.2124
C01745=29.931,-95.359,61.359,179.8441,-0.0009,-10242.5741
C01746=24.496,-96.092,61.037,177.6795,-0.8285,-10245.6986
C01747=19.672,-94.474,60.719,176.4586,-3.3893,-10248.2376
C01748=16.396,-90.884,60.330,177.7605,-7.7070,-10249.7735
